   1:  PR[91,3] = PR[90,3] + 20.865;
   1:L PR[91] R[100]mm/sec CNT100;
   1:  PR[91,1] = PR[90,1] + -32.323;
   1:  PR[91,2] = PR[90,2] + 9.963;
   1:  PR[91,3] = PR[90,3] + 20.871;
   1:L PR[91] R[100]mm/sec CNT100;
   1:  PR[91,1] = PR[90,1] + -32.788;
   1:  PR[91,2] = PR[90,2] + 9.239;
   1:  PR[91,3] = PR[90,3] + 20.877;
   1:L PR[91] R[100]mm/sec CNT100;
   1:  PR[91,1] = PR[90,1] + -33.216;
   1:  PR[91,2] = PR[90,2] + 8.495;
   1:  PR[91,3] = PR[90,3] + 20.883;
   1:L PR[91] R[100]mm/sec CNT100;
   1:  PR[91,1] = PR[90,1] + -33.606;
   1:  PR[91,2] = PR[90,2] + 7.735;
   1:  PR[91,3] = PR[90,3] + 20.889;
   1:L PR[91] R[100]mm/sec CNT100;
   1:  PR[91,1] = PR[90,1] + -33.957;
   1:  PR[91,2] = PR[90,2] + 6.963;
   1:  PR[91,3] = PR[90,3] + 20.895;
   1:L PR[91] R[100]mm/sec CNT100;
   1:  PR[91,1] = PR[90,1] + -34.268;
   1:  PR[91,2] = PR[90,2] + 6.184;
   1:  PR[91,3] = PR[90,3] + 20.901;
   1:L PR[91] R[100]mm/sec CNT100;
   1:  PR[91,1] = PR[90,1] + -34.538;
   1:  PR[91,2] = PR[90,2] + 5.400;
   1:  PR[91,3] = PR[90,3] + 20.907;
   1:L PR[91] R[100]mm/sec CNT100;
   1:  PR[91,1] = PR[90,1] + -34.767;
   1:  PR[91,2] = PR[90,2] + 4.609;
   1:  PR[91,3] = PR[90,3] + 20.913;
   1:L PR[91] R[100]mm/sec CNT100;
   1:  PR[91,1] = PR[90,1] + -34.955;
   1:  PR[91,2] = PR[90,2] + 3.810;
   1:  PR[91,3] = PR[90,3] + 20.918;
   1:L PR[91] R[100]mm/sec CNT100;
   1:  PR[91,1] = PR[90,1] + -35.101;
   1:  PR[91,2] = PR[90,2] + 2.999;
   1:  PR[91,3] = PR[90,3] + 20.924;
   1:L PR[91] R[100]mm/sec CNT100;
   1:  PR[91,1] = PR[90,1] + -35.206;
   1:  PR[91,2] = PR[90,2] + 2.168;
   1:  PR[91,3] = PR[90,3] + 20.930;
   1:L PR[91] R[100]mm/sec CNT100;
   1:  PR[91,1] = PR[90,1] + -35.270;
   1:  PR[91,2] = PR[90,2] + 1.312;
   1:  PR[91,3] = PR[90,3] + 20.936;
   1:L PR[91] R[100]mm/sec CNT100;
   1:  PR[91,1] = PR[90,1] + -35.294;
   1:  PR[91,2] = PR[90,2] + 0.428;
   1:  PR[91,3] = PR[90,3] + 20.942;
   1:L PR[91] R[100]mm/sec CNT100;
   1:  PR[91,1] = PR[90,1] + -35.270;
   1:  PR[91,2] = PR[90,2] + -0.456;
   1:  PR[91,3] = PR[90,3] + 20.948;
   1:L PR[91] R[100]mm/sec CNT100;
   1:  PR[91,1] = PR[90,1] + -35.206;
   1:  PR[91,2] = PR[90,2] + -1.313;
   1:  PR[91,3] = PR[90,3] + 20.954;
   1:L PR[91] R[100]mm/sec CNT100;
   1:  PR[91,1] = PR[90,1] + -35.101;
   1:  PR[91,2] = PR[90,2] + -2.144;
   1:  PR[91,3] = PR[90,3] + 20.960;
   1:L PR[91] R[100]mm/sec CNT100;
   1:  PR[91,1] = PR[90,1] + -34.955;
   1:  PR[91,2] = PR[90,2] + -2.955;
   1:  PR[91,3] = PR[90,3] + 20.966;
   1:L PR[91] R[100]mm/sec CNT100;
   1:  PR[91,1] = PR[90,1] + -34.767;
   1:  PR[91,2] = PR[90,2] + -3.754;
   1:  PR[91,3] = PR[90,3] + 20.972;
   1:L PR[91] R[100]mm/sec CNT100;
   1:  PR[91,1] = PR[90,1] + -34.538;
   1:  PR[91,2] = PR[90,2] + -4.545;
   1:  PR[91,3] = PR[90,3] + 20.978;
   1:L PR[91] R[100]mm/sec CNT100;
   1:  PR[91,1] = PR[90,1] + -34.268;
   1:  PR[91,2] = PR[90,2] + -5.329;
   1:  PR[91,3] = PR[90,3] + 20.984;
   1:L PR[91] R[100]mm/sec CNT100;
   1:  PR[91,1] = PR[90,1] + -33.956;
   1:  PR[91,2] = PR[90,2] + -6.108;
   1:  PR[91,3] = PR[90,3] + 20.989;
   1:L PR[91] R[100]mm/sec CNT100;
   1:  PR[91,1] = PR[90,1] + -33.606;
   1:  PR[91,2] = PR[90,2] + -6.880;
   1:  PR[91,3] = PR[90,3] + 20.995;
   1:L PR[91] R[100]mm/sec CNT100;
   1:  PR[91,1] = PR[90,1] + -33.216;
   1:  PR[91,2] = PR[90,2] + -7.640;
   1:  PR[91,3] = PR[90,3] + 21.001;
   1:L PR[91] R[100]mm/sec CNT100;
   1:  PR[91,1] = PR[90,1] + -32.788;
   1:  PR[91,2] = PR[90,2] + -8.384;
   1:  PR[91,3] = PR[90,3] + 21.007;
   1:L PR[91] R[100]mm/sec CNT100;
   1:  PR[91,1] = PR[90,1] + -32.323;
   1:  PR[91,2] = PR[90,2] + -9.108;
   1:  PR[91,3] = PR[90,3] + 21.013;
   1:L PR[91] R[100]mm/sec CNT100;
   1:  PR[91,1] = PR[90,1] + -31.822;
   1:  PR[91,2] = PR[90,2] + -9.809;
   1:  PR[91,3] = PR[90,3] + 21.019;
   1:L PR[91] R[100]mm/sec CNT100;
   1:  PR[91,1] = PR[90,1] + -31.285;
   1:  PR[91,2] = PR[90,2] + -10.485;
   1:  PR[91,3] = PR[90,3] + 21.026;
   1:L PR[91] R[100]mm/sec CNT100;
   1:  PR[91,1] = PR[90,1] + -30.715;
   1:  PR[91,2] = PR[90,2] + -11.134;
   1:  PR[91,3] = PR[90,3] + 21.032;
   1:L PR[91] R[100]mm/sec CNT100;
   1:  PR[91,1] = PR[90,1] + -30.107;
   1:  PR[91,2] = PR[90,2] + -11.756;
   1:  PR[91,3] = PR[90,3] + 21.038;
   1:L PR[91] R[100]mm/sec CNT100;
   1:  PR[91,1] = PR[90,1] + -29.466;
   1:  PR[91,2] = PR[90,2] + -12.350;
   1:  PR[91,3] = PR[90,3] + 21.044;
   1:L PR[91] R[100]mm/sec CNT100;
   1:  PR[91,1] = PR[90,1] + -28.795;
   1:  PR[91,2] = PR[90,2] + -12.914;
   1:  PR[91,3] = PR[90,3] + 21.050;
   1:L PR[91] R[100]mm/sec CNT100;
   1:  PR[91,1] = PR[90,1] + -28.093;
   1:  PR[91,2] = PR[90,2] + -13.447;
   1:  PR[91,3] = PR[90,3] + 21.056;
   1:L PR[91] R[100]mm/sec CNT100;
   1:  PR[91,1] = PR[90,1] + -27.361;
   1:  PR[91,2] = PR[90,2] + -13.949;
   1:  PR[91,3] = PR[90,3] + 21.062;
   1:L PR[91] R[100]mm/sec CNT100;
   1:  PR[91,1] = PR[90,1] + -27.042;
   1:  PR[91,2] = PR[90,2] + -14.147;
   1:  PR[91,3] = PR[90,3] + 21.069;
   1:L PR[91] R[100]mm/sec CNT100;
   1:  PR[91,1] = PR[90,1] + -26.605;
   1:  PR[91,2] = PR[90,2] + -14.416;
   1:  PR[91,3] = PR[90,3] + 21.071;
   1:L PR[91] R[100]mm/sec CNT100;
   1:  PR[91,1] = PR[90,1] + -25.820;
   1:  PR[91,2] = PR[90,2] + -14.850;
   1:  PR[91,3] = PR[90,3] + 21.075;
   1:L PR[91] R[100]mm/sec CNT100;
   1:  PR[91,1] = PR[90,1] + -25.013;
   1:  PR[91,2] = PR[90,2] + -15.247;
   1:  PR[91,3] = PR[90,3] + 21.081;
   1:L PR[91] R[100]mm/sec CNT100;
   1:  PR[91,1] = PR[90,1] + -24.202;
   1:  PR[91,2] = PR[90,2] + -15.599;
   1:  PR[91,3] = PR[90,3] + 21.087;
   1:L PR[91] R[100]mm/sec CNT100;
   1:  PR[91,1] = PR[90,1] + -23.226;
   1:  PR[91,2] = PR[90,2] + -15.963;
   1:  PR[91,3] = PR[90,3] + 21.094;
   1:L PR[91] R[100]mm/sec CNT100;
   1:  PR[91,1] = PR[90,1] + -22.273;
   1:  PR[91,2] = PR[90,2] + -16.262;
   1:  PR[91,3] = PR[90,3] + 21.101;
   1:L PR[91] R[100]mm/sec CNT100;
   1:  PR[91,1] = PR[90,1] + -21.780;
   1:  PR[91,2] = PR[90,2] + -16.396;
   1:  PR[91,3] = PR[90,3] + 21.108;
   1:L PR[91] R[100]mm/sec CNT100;
   1:  PR[91,1] = PR[90,1] + -20.956;
   1:  PR[91,2] = PR[90,2] + -16.588;
   1:  PR[91,3] = PR[90,3] + 21.112;
   1:L PR[91] R[100]mm/sec CNT100;
   1:  PR[91,1] = PR[90,1] + -20.130;
   1:  PR[91,2] = PR[90,2] + -16.744;
   1:  PR[91,3] = PR[90,3] + 21.118;
   1:L PR[91] R[100]mm/sec CNT100;
   1:  PR[91,1] = PR[90,1] + -19.301;
   1:  PR[91,2] = PR[90,2] + -16.862;
   1:  PR[91,3] = PR[90,3] + 21.124;
   1:L PR[91] R[100]mm/sec CNT100;
   1:  PR[91,1] = PR[90,1] + -18.404;
   1:  PR[91,2] = PR[90,2] + -16.950;
   1:  PR[91,3] = PR[90,3] + 21.129;
   1:L PR[91] R[100]mm/sec CNT100;
   1:  PR[91,1] = PR[90,1] + -17.474;
   1:  PR[91,2] = PR[90,2] + -16.997;
   1:  PR[91,3] = PR[90,3] + 21.136;
   1:L PR[91] R[100]mm/sec CNT100;
   1:  PR[91,1] = PR[90,1] + -16.945;
   1:  PR[91,2] = PR[90,2] + -17.001;
   1:  PR[91,3] = PR[90,3] + 21.142;
   1:L PR[91] R[100]mm/sec CNT100;
   1:  PR[91,1] = PR[90,1] + -16.543;
   1:  PR[91,3] = PR[90,3] + 21.146;
   1:L PR[91] R[100]mm/sec CNT100;
   1:  PR[91,1] = PR[90,1] + -15.605;
   1:  PR[91,2] = PR[90,2] + -16.959;
   1:  PR[91,3] = PR[90,3] + 21.149;
   1:L PR[91] R[100]mm/sec CNT100;
   1:  PR[91,1] = PR[90,1] + -14.668;
   1:  PR[91,2] = PR[90,2] + -16.872;
   1:  PR[91,3] = PR[90,3] + 21.156;
   1:L PR[91] R[100]mm/sec CNT100;
   1:  PR[91,1] = PR[90,1] + -13.745;
   1:  PR[91,2] = PR[90,2] + -16.743;
   1:  PR[91,3] = PR[90,3] + 21.162;
   1:L PR[91] R[100]mm/sec CNT100;
   1:  PR[91,1] = PR[90,1] + -12.925;
   1:  PR[91,2] = PR[90,2] + -16.592;
   1:  PR[91,3] = PR[90,3] + 21.169;
   1:L PR[91] R[100]mm/sec CNT100;
   1:  PR[91,1] = PR[90,1] + -11.875;
   1:  PR[91,2] = PR[90,2] + -16.344;
   1:  PR[91,3] = PR[90,3] + 21.175;
   1:L PR[91] R[100]mm/sec CNT100;
   1:  PR[91,1] = PR[90,1] + -11.166;
   1:  PR[91,2] = PR[90,2] + -16.141;
   1:  PR[91,3] = PR[90,3] + 21.182;
   1:L PR[91] R[100]mm/sec CNT100;
   1:  PR[91,1] = PR[90,1] + -10.545;
   1:  PR[91,2] = PR[90,2] + -15.938;
   1:  PR[91,3] = PR[90,3] + 21.187;
   1:L PR[91] R[100]mm/sec CNT100;
   1:  PR[91,1] = PR[90,1] + -9.970;
   1:  PR[91,2] = PR[90,2] + -15.731;
   1:  PR[91,3] = PR[90,3] + 21.192;
   1:L PR[91] R[100]mm/sec CNT100;
   1:  PR[91,1] = PR[90,1] + -9.341;
   1:  PR[91,2] = PR[90,2] + -15.480;
   1:  PR[91,3] = PR[90,3] + 21.196;
   1:L PR[91] R[100]mm/sec CNT100;
   1:  PR[91,1] = PR[90,1] + -8.803;
   1:  PR[91,2] = PR[90,2] + -15.246;
   1:  PR[91,3] = PR[90,3] + 21.201;
   1:L PR[91] R[100]mm/sec CNT100;
   1:  PR[91,1] = PR[90,1] + -8.183;
   1:  PR[91,2] = PR[90,2] + -14.951;
   1:  PR[91,3] = PR[90,3] + 21.205;
   1:L PR[91] R[100]mm/sec CNT100;
   1:  PR[91,1] = PR[90,1] + -7.109;
   1:  PR[91,2] = PR[90,2] + -14.372;
   1:  PR[91,3] = PR[90,3] + 21.210;
   1:L PR[91] R[100]mm/sec CNT100;
   1:  PR[91,1] = PR[90,1] + -6.488;
   1:  PR[91,2] = PR[90,2] + -13.995;
   1:  PR[91,3] = PR[90,3] + 21.219;
   1:L PR[91] R[100]mm/sec CNT100;
   1:  PR[91,1] = PR[90,1] + -5.527;
   1:  PR[91,2] = PR[90,2] + -13.342;
   1:  PR[91,3] = PR[90,3] + 21.224;
   1:L PR[91] R[100]mm/sec CNT100;
   1:  PR[91,1] = PR[90,1] + -4.920;
   1:  PR[91,2] = PR[90,2] + -12.883;
   1:  PR[91,3] = PR[90,3] + 21.232;
   1:L PR[91] R[100]mm/sec CNT100;
   1:  PR[91,1] = PR[90,1] + -4.075;
   1:  PR[91,2] = PR[90,2] + -12.171;
   1:  PR[91,3] = PR[90,3] + 21.237;
   1:L PR[91] R[100]mm/sec CNT100;
   1:  PR[91,1] = PR[90,1] + -3.306;
   1:  PR[91,2] = PR[90,2] + -11.437;
   1:  PR[91,3] = PR[90,3] + 21.245;
   1:L PR[91] R[100]mm/sec CNT100;
   1:  PR[91,1] = PR[90,1] + -2.752;
   1:  PR[91,2] = PR[90,2] + -10.852;
   1:  PR[91,3] = PR[90,3] + 21.253;
   1:L PR[91] R[100]mm/sec CNT100;
   1:  PR[91,1] = PR[90,1] + -2.351;
   1:  PR[91,2] = PR[90,2] + -10.384;
   1:  PR[91,3] = PR[90,3] + 21.258;
   1:L PR[91] R[100]mm/sec CNT100;
   1:  PR[91,1] = PR[90,1] + -2.018;
   1:  PR[91,2] = PR[90,2] + -10.037;
   1:  PR[91,3] = PR[90,3] + 21.263;
   1:L PR[91] R[100]mm/sec CNT100;
   1:  PR[91,1] = PR[90,1] + -1.614;
   1:  PR[91,2] = PR[90,2] + -9.738;
   1:  PR[91,3] = PR[90,3] + 21.266;
   1:L PR[91] R[100]mm/sec CNT100;
   1:  PR[91,1] = PR[90,1] + -1.170;
   1:  PR[91,2] = PR[90,2] + -9.512;
   1:  PR[91,3] = PR[90,3] + 21.269;
   1:L PR[91] R[100]mm/sec CNT100;
   1:  PR[91,1] = PR[90,1] + -0.694;
   1:  PR[91,2] = PR[90,2] + -9.365;
   1:  PR[91,3] = PR[90,3] + 21.273;
   1:L PR[91] R[100]mm/sec CNT100;
   1:  PR[91,1] = PR[90,1] + -0.199;
   1:  PR[91,2] = PR[90,2] + -9.306;
   1:  PR[91,3] = PR[90,3] + 21.276;
   1:L PR[91] R[100]mm/sec CNT100;
   1:  PR[91] = PR[90];
   1:  PR[91,1] = PR[90,1] + 0.421;
   1:  PR[91,2] = PR[90,2] + -10.128;
   1:  PR[91,3] = PR[90,3] + 22.610;
   1:L PR[91] R[100]mm/sec CNT100;
   1:  PR[91,1] = PR[90,1] + 0.906;
   1:  PR[91,2] = PR[90,2] + -10.267;
   1:  PR[91,3] = PR[90,3] + 21.284;
   1:L PR[91] R[100]mm/sec CNT100;
   1:  PR[91,1] = PR[90,1] + 1.365;
   1:  PR[91,2] = PR[90,2] + -10.492;
   1:  PR[91,3] = PR[90,3] + 21.287;
   1:L PR[91] R[100]mm/sec CNT100;
   1:  PR[91,1] = PR[90,1] + 1.785;
   1:  PR[91,2] = PR[90,2] + -10.796;
   1:  PR[91,3] = PR[90,3] + 21.291;
   1:L PR[91] R[100]mm/sec CNT100;
   1:  PR[91,1] = PR[90,1] + 2.627;
   1:  PR[91,2] = PR[90,2] + -11.664;
   1:  PR[91,3] = PR[90,3] + 21.294;
   1:L PR[91] R[100]mm/sec CNT100;
   1:  PR[91,1] = PR[90,1] + 3.330;
   1:  PR[91,2] = PR[90,2] + -12.323;
   1:  PR[91,3] = PR[90,3] + 21.303;
   1:L PR[91] R[100]mm/sec CNT100;
   1:  PR[91,1] = PR[90,1] + 4.018;
   1:  PR[91,2] = PR[90,2] + -12.904;
   1:  PR[91,3] = PR[90,3] + 21.310;
   1:L PR[91] R[100]mm/sec CNT100;
   1:  PR[91,1] = PR[90,1] + 4.792;
   1:  PR[91,2] = PR[90,2] + -13.492;
   1:  PR[91,3] = PR[90,3] + 21.316;
   1:L PR[91] R[100]mm/sec CNT100;
   1:  PR[91,1] = PR[90,1] + 5.634;
   1:  PR[91,2] = PR[90,2] + -14.062;
   1:  PR[91,3] = PR[90,3] + 21.323;
   1:L PR[91] R[100]mm/sec CNT100;
   1:  PR[91,1] = PR[90,1] + 6.385;
   1:  PR[91,2] = PR[90,2] + -14.517;
   1:  PR[91,3] = PR[90,3] + 21.331;
   1:L PR[91] R[100]mm/sec CNT100;
   1:  PR[91,1] = PR[90,1] + 7.324;
   1:  PR[91,2] = PR[90,2] + -15.021;
   1:  PR[91,3] = PR[90,3] + 21.337;
   1:L PR[91] R[100]mm/sec CNT100;
   1:  PR[91,1] = PR[90,1] + 8.080;
   1:  PR[91,2] = PR[90,2] + -15.379;
   1:  PR[91,3] = PR[90,3] + 21.344;
   1:L PR[91] R[100]mm/sec CNT100;
   1:  PR[91,1] = PR[90,1] + 9.117;
   1:  PR[91,2] = PR[90,2] + -15.808;
   1:  PR[91,3] = PR[90,3] + 21.350;
   1:L PR[91] R[100]mm/sec CNT100;
   1:  PR[91,1] = PR[90,1] + 9.860;
   1:  PR[91,2] = PR[90,2] + -16.074;
   1:  PR[91,3] = PR[90,3] + 21.358;
   1:L PR[91] R[100]mm/sec CNT100;
   1:  PR[91,1] = PR[90,1] + 10.982;
   1:  PR[91,2] = PR[90,2] + -16.413;
   1:  PR[91,3] = PR[90,3] + 21.364;
   1:L PR[91] R[100]mm/sec CNT100;
   1:  PR[91,1] = PR[90,1] + 12.190;
   1:  PR[91,2] = PR[90,2] + -16.698;
   1:  PR[91,3] = PR[90,3] + 21.372;
   1:L PR[91] R[100]mm/sec CNT100;
   1:  PR[91,1] = PR[90,1] + 12.901;
   1:  PR[91,2] = PR[90,2] + -16.830;
   1:  PR[91,3] = PR[90,3] + 21.381;
   1:L PR[91] R[100]mm/sec CNT100;
   1:  PR[91,1] = PR[90,1] + 13.574;
   1:  PR[91,2] = PR[90,2] + -16.929;
   1:  PR[91,3] = PR[90,3] + 21.386;
   1:L PR[91] R[100]mm/sec CNT100;
   1:  PR[91,1] = PR[90,1] + 14.840;
   1:  PR[91,2] = PR[90,2] + -17.053;
   1:  PR[91,3] = PR[90,3] + 21.391;
   1:L PR[91] R[100]mm/sec CNT100;
   1:  PR[91,1] = PR[90,1] + 16.006;
   1:  PR[91,2] = PR[90,2] + -17.097;
   1:  PR[91,3] = PR[90,3] + 21.400;
   1:L PR[91] R[100]mm/sec CNT100;
   1:  PR[91,1] = PR[90,1] + 16.711;
   1:  PR[91,2] = PR[90,2] + -17.091;
   1:  PR[91,3] = PR[90,3] + 21.409;
   1:L PR[91] R[100]mm/sec CNT100;
   1:  PR[91,1] = PR[90,1] + 17.506;
   1:  PR[91,2] = PR[90,2] + -17.054;
   1:  PR[91,3] = PR[90,3] + 21.414;
   1:L PR[91] R[100]mm/sec CNT100;
   1:  PR[91,1] = PR[90,1] + 18.499;
   1:  PR[91,2] = PR[90,2] + -16.963;
   1:  PR[91,3] = PR[90,3] + 21.419;
   1:L PR[91] R[100]mm/sec CNT100;
   1:  PR[91,1] = PR[90,1] + 19.377;
   1:  PR[91,2] = PR[90,2] + -16.840;
   1:  PR[91,3] = PR[90,3] + 21.426;
   1:L PR[91] R[100]mm/sec CNT100;
   1:  PR[91,1] = PR[90,1] + 20.291;
   1:  PR[91,2] = PR[90,2] + -16.668;
   1:  PR[91,3] = PR[90,3] + 21.433;
   1:L PR[91] R[100]mm/sec CNT100;
   1:  PR[91,1] = PR[90,1] + 21.192;
   1:  PR[91,2] = PR[90,2] + -16.455;
   1:  PR[91,3] = PR[90,3] + 21.439;
   1:L PR[91] R[100]mm/sec CNT100;
   1:  PR[91,1] = PR[90,1] + 22.077;
   1:  PR[91,2] = PR[90,2] + -16.200;
   1:  PR[91,3] = PR[90,3] + 21.446;
   1:L PR[91] R[100]mm/sec CNT100;
   1:  PR[91,1] = PR[90,1] + 22.945;
   1:  PR[91,2] = PR[90,2] + -15.905;
   1:  PR[91,3] = PR[90,3] + 21.453;
   1:L PR[91] R[100]mm/sec CNT100;
   1:  PR[91,1] = PR[90,1] + 23.794;
   1:  PR[91,2] = PR[90,2] + -15.572;
   1:  PR[91,3] = PR[90,3] + 21.459;
   1:L PR[91] R[100]mm/sec CNT100;
   1:  PR[91,1] = PR[90,1] + 24.595;
   1:  PR[91,2] = PR[90,2] + -15.214;
   1:  PR[91,3] = PR[90,3] + 21.466;
   1:L PR[91] R[100]mm/sec CNT100;
   1:  PR[91,1] = PR[90,1] + 25.352;
   1:  PR[91,2] = PR[90,2] + -14.833;
   1:  PR[91,3] = PR[90,3] + 21.472;
   1:L PR[91] R[100]mm/sec CNT100;
   1:  PR[91,1] = PR[90,1] + 26.092;
   1:  PR[91,2] = PR[90,2] + -14.417;
   1:  PR[91,3] = PR[90,3] + 21.478;
   1:L PR[91] R[100]mm/sec CNT100;
   1:  PR[91,1] = PR[90,1] + 26.814;
   1:  PR[91,2] = PR[90,2] + -13.968;
   1:  PR[91,3] = PR[90,3] + 21.484;
   1:L PR[91] R[100]mm/sec CNT100;
   1:  PR[91,1] = PR[90,1] + 27.516;
   1:  PR[91,2] = PR[90,2] + -13.485;
   1:  PR[91,3] = PR[90,3] + 21.490;
   1:L PR[91] R[100]mm/sec CNT100;
   1:  PR[91,1] = PR[90,1] + 28.196;
   1:  PR[91,2] = PR[90,2] + -12.969;
   1:  PR[91,3] = PR[90,3] + 21.496;
   1:L PR[91] R[100]mm/sec CNT100;
   1:  PR[91,1] = PR[90,1] + 28.852;
   1:  PR[91,2] = PR[90,2] + -12.420;
   1:  PR[91,3] = PR[90,3] + 21.502;
   1:L PR[91] R[100]mm/sec CNT100;
   1:  PR[91,1] = PR[90,1] + 29.481;
   1:  PR[91,2] = PR[90,2] + -11.840;
   1:  PR[91,3] = PR[90,3] + 21.508;
   1:L PR[91] R[100]mm/sec CNT100;
   1:  PR[91,1] = PR[90,1] + 30.083;
   1:  PR[91,2] = PR[90,2] + -11.228;
   1:  PR[91,3] = PR[90,3] + 21.514;
   1:L PR[91] R[100]mm/sec CNT100;
   1:  PR[91,1] = PR[90,1] + 30.665;
   1:  PR[91,2] = PR[90,2] + -10.571;
   1:  PR[91,3] = PR[90,3] + 21.521;
   1:L PR[91] R[100]mm/sec CNT100;
   1:  PR[91,1] = PR[90,1] + 31.212;
   1:  PR[91,2] = PR[90,2] + -9.887;
   1:  PR[91,3] = PR[90,3] + 21.527;
   1:L PR[91] R[100]mm/sec CNT100;
   1:  PR[91,1] = PR[90,1] + 31.723;
   1:  PR[91,2] = PR[90,2] + -9.178;
   1:  PR[91,3] = PR[90,3] + 21.533;
   1:L PR[91] R[100]mm/sec CNT100;
   1:  PR[91,1] = PR[90,1] + 32.197;
   1:  PR[91,2] = PR[90,2] + -8.448;
   1:  PR[91,3] = PR[90,3] + 21.539;
   1:L PR[91] R[100]mm/sec CNT100;
   1:  PR[91,1] = PR[90,1] + 32.633;
   1:  PR[91,2] = PR[90,2] + -7.699;
   1:  PR[91,3] = PR[90,3] + 21.545;
   1:L PR[91] R[100]mm/sec CNT100;
   1:  PR[91,1] = PR[90,1] + 33.030;
   1:  PR[91,2] = PR[90,2] + -6.937;
   1:  PR[91,3] = PR[90,3] + 21.552;
   1:L PR[91] R[100]mm/sec CNT100;
   1:  PR[91,1] = PR[90,1] + 33.388;
   1:  PR[91,2] = PR[90,2] + -6.164;
   1:  PR[91,3] = PR[90,3] + 21.558;
   1:L PR[91] R[100]mm/sec CNT100;
   1:  PR[91,1] = PR[90,1] + 33.704;
   1:  PR[91,2] = PR[90,2] + -5.385;
   1:  PR[91,3] = PR[90,3] + 21.564;
   1:L PR[91] R[100]mm/sec CNT100;
   1:  PR[91,1] = PR[90,1] + 33.979;
   1:  PR[91,2] = PR[90,2] + -4.600;
   1:  PR[91,3] = PR[90,3] + 21.570;
   1:L PR[91] R[100]mm/sec CNT100;
   1:  PR[91,1] = PR[90,1] + 34.212;
   1:  PR[91,2] = PR[90,2] + -3.806;
   1:  PR[91,3] = PR[90,3] + 21.576;
   1:L PR[91] R[100]mm/sec CNT100;
   1:  PR[91,1] = PR[90,1] + 34.403;
   1:  PR[91,2] = PR[90,2] + -3.001;
   1:  PR[91,3] = PR[90,3] + 21.582;
   1:L PR[91] R[100]mm/sec CNT100;
   1:  PR[91,1] = PR[90,1] + 34.552;
   1:  PR[91,2] = PR[90,2] + -2.180;
   1:  PR[91,3] = PR[90,3] + 21.588;
   1:L PR[91] R[100]mm/sec CNT100;
   1:  PR[91,1] = PR[90,1] + 34.659;
   1:  PR[91,2] = PR[90,2] + -1.338;
   1:  PR[91,3] = PR[90,3] + 21.594;
   1:L PR[91] R[100]mm/sec CNT100;
   1:  PR[91,1] = PR[90,1] + 34.724;
   1:  PR[91,2] = PR[90,2] + -0.470;
   1:  PR[91,3] = PR[90,3] + 21.600;
   1:L PR[91] R[100]mm/sec CNT100;
   1:  PR[91,1] = PR[90,1] + 34.745;
   1:  PR[91,2] = PR[90,2] + 0.428;
   1:  PR[91,3] = PR[90,3] + 21.606;
   1:L PR[91] R[100]mm/sec CNT100;
   1:  PR[91,1] = PR[90,1] + 34.724;
   1:  PR[91,2] = PR[90,2] + 1.325;
   1:  PR[91,3] = PR[90,3] + 21.612;
   1:L PR[91] R[100]mm/sec CNT100;
   1:  PR[91,1] = PR[90,1] + 34.659;
   1:  PR[91,2] = PR[90,2] + 2.193;
   1:  PR[91,3] = PR[90,3] + 21.619;
   1:L PR[91] R[100]mm/sec CNT100;
   1:  PR[91,1] = PR[90,1] + 34.552;
   1:  PR[91,2] = PR[90,2] + 3.035;
   1:  PR[91,3] = PR[90,3] + 21.625;
   1:L PR[91] R[100]mm/sec CNT100;
   1:  PR[91,1] = PR[90,1] + 34.403;
   1:  PR[91,2] = PR[90,2] + 3.856;
   1:  PR[91,3] = PR[90,3] + 21.631;
   1:L PR[91] R[100]mm/sec CNT100;
   1:  PR[91,1] = PR[90,1] + 34.212;
   1:  PR[91,2] = PR[90,2] + 4.661;
   1:  PR[91,3] = PR[90,3] + 21.637;
   1:L PR[91] R[100]mm/sec CNT100;
   1:  PR[91,1] = PR[90,1] + 33.979;
   1:  PR[91,2] = PR[90,2] + 5.455;
   1:  PR[91,3] = PR[90,3] + 21.643;
   1:L PR[91] R[100]mm/sec CNT100;
   1:  PR[91,1] = PR[90,1] + 33.704;
   1:  PR[91,2] = PR[90,2] + 6.241;
   1:  PR[91,3] = PR[90,3] + 21.649;
   1:L PR[91] R[100]mm/sec CNT100;
   1:  PR[91,1] = PR[90,1] + 33.388;
   1:  PR[91,2] = PR[90,2] + 7.019;
   1:  PR[91,3] = PR[90,3] + 21.655;
   1:L PR[91] R[100]mm/sec CNT100;
   1:  PR[91,1] = PR[90,1] + 33.030;
   1:  PR[91,2] = PR[90,2] + 7.792;
   1:  PR[91,3] = PR[90,3] + 21.661;
   1:L PR[91] R[100]mm/sec CNT100;
   1:  PR[91,1] = PR[90,1] + 32.633;
   1:  PR[91,2] = PR[90,2] + 8.554;
   1:  PR[91,3] = PR[90,3] + 21.667;
   1:L PR[91] R[100]mm/sec CNT100;
   1:  PR[91,1] = PR[90,1] + 32.197;
   1:  PR[91,2] = PR[90,2] + 9.303;
   1:  PR[91,3] = PR[90,3] + 21.673;
   1:L PR[91] R[100]mm/sec CNT100;
   1:  PR[91,1] = PR[90,1] + 31.723;
   1:  PR[91,2] = PR[90,2] + 10.033;
   1:  PR[91,3] = PR[90,3] + 21.679;
   1:L PR[91] R[100]mm/sec CNT100;
   1:  PR[91,1] = PR[90,1] + 31.212;
   1:  PR[91,2] = PR[90,2] + 10.742;
   1:  PR[91,3] = PR[90,3] + 21.685;
   1:L PR[91] R[100]mm/sec CNT100;
   1:  PR[91,1] = PR[90,1] + 30.665;
   1:  PR[91,2] = PR[90,2] + 11.426;
   1:  PR[91,3] = PR[90,3] + 21.691;
   1:L PR[91] R[100]mm/sec CNT100;
   1:  PR[91,1] = PR[90,1] + 30.081;
   1:  PR[91,2] = PR[90,2] + 12.086;
   1:  PR[91,3] = PR[90,3] + 21.698;
   1:L PR[91] R[100]mm/sec CNT100;
   1:  PR[91,1] = PR[90,1] + 29.481;
   1:  PR[91,2] = PR[90,2] + 12.695;
   1:  PR[91,3] = PR[90,3] + 21.704;
   1:L PR[91] R[100]mm/sec CNT100;
   1:  PR[91,1] = PR[90,1] + 28.852;
   1:  PR[91,2] = PR[90,2] + 13.276;
   1:  PR[91,3] = PR[90,3] + 21.710;
   1:L PR[91] R[100]mm/sec CNT100;
   1:  PR[91,1] = PR[90,1] + 28.196;
   1:  PR[91,2] = PR[90,2] + 13.824;
   1:  PR[91,3] = PR[90,3] + 21.716;
   1:L PR[91] R[100]mm/sec CNT100;
   1:  PR[91,1] = PR[90,1] + 27.515;
   1:  PR[91,2] = PR[90,2] + 14.341;
   1:  PR[91,3] = PR[90,3] + 21.722;
   1:L PR[91] R[100]mm/sec CNT100;
   1:  PR[91,1] = PR[90,1] + 27.184;
   1:  PR[91,2] = PR[90,2] + 14.571;
   1:  PR[91,3] = PR[90,3] + 21.728;
   1:L PR[91] R[100]mm/sec CNT100;
   1:  PR[91,1] = PR[90,1] + 26.815;
   1:  PR[91,2] = PR[90,2] + 14.822;
   1:  PR[91,3] = PR[90,3] + 21.731;
   1:L PR[91] R[100]mm/sec CNT100;
   1:  PR[91,1] = PR[90,1] + 26.092;
   1:  PR[91,2] = PR[90,2] + 15.272;
   1:  PR[91,3] = PR[90,3] + 21.734;
   1:L PR[91] R[100]mm/sec CNT100;
   1:  PR[91,1] = PR[90,1] + 25.352;
   1:  PR[91,2] = PR[90,2] + 15.688;
   1:  PR[91,3] = PR[90,3] + 21.740;
   1:L PR[91] R[100]mm/sec CNT100;
   1:  PR[91,1] = PR[90,1] + 24.595;
   1:  PR[91,2] = PR[90,2] + 16.069;
   1:  PR[91,3] = PR[90,3] + 21.746;
   1:L PR[91] R[100]mm/sec CNT100;
   1:  PR[91,1] = PR[90,1] + 23.794;
   1:  PR[91,2] = PR[90,2] + 16.428;
   1:  PR[91,3] = PR[90,3] + 21.752;
   1:L PR[91] R[100]mm/sec CNT100;
   1:  PR[91,1] = PR[90,1] + 22.944;
   1:  PR[91,2] = PR[90,2] + 16.761;
   1:  PR[91,3] = PR[90,3] + 21.759;
   1:L PR[91] R[100]mm/sec CNT100;
   1:  PR[91,1] = PR[90,1] + 22.377;
   1:  PR[91,2] = PR[90,2] + 16.955;
   1:  PR[91,3] = PR[90,3] + 21.765;
   1:L PR[91] R[100]mm/sec CNT100;
   1:  PR[91,1] = PR[90,1] + 22.078;
   1:  PR[91,2] = PR[90,2] + 17.055;
   1:  PR[91,3] = PR[90,3] + 21.770;
   1:L PR[91] R[100]mm/sec CNT100;
   1:  PR[91,1] = PR[90,1] + 21.194;
   1:  PR[91,2] = PR[90,2] + 17.309;
   1:  PR[91,3] = PR[90,3] + 21.772;
   1:L PR[91] R[100]mm/sec CNT100;
   1:  PR[91,1] = PR[90,1] + 20.105;
   1:  PR[91,2] = PR[90,2] + 17.560;
   1:  PR[91,3] = PR[90,3] + 21.778;
   1:L PR[91] R[100]mm/sec CNT100;
   1:  PR[91,1] = PR[90,1] + 19.377;
   1:  PR[91,2] = PR[90,2] + 17.695;
   1:  PR[91,3] = PR[90,3] + 21.786;
   1:L PR[91] R[100]mm/sec CNT100;
   1:  PR[91,1] = PR[90,1] + 18.499;
   1:  PR[91,2] = PR[90,2] + 17.818;
   1:  PR[91,3] = PR[90,3] + 21.792;
   1:L PR[91] R[100]mm/sec CNT100;
   1:  PR[91,1] = PR[90,1] + 17.506;
   1:  PR[91,2] = PR[90,2] + 17.909;
   1:  PR[91,3] = PR[90,3] + 21.798;
   1:L PR[91] R[100]mm/sec CNT100;
   1:  PR[91,1] = PR[90,1] + 16.710;
   1:  PR[91,2] = PR[90,2] + 17.946;
   1:  PR[91,3] = PR[90,3] + 21.805;
   1:L PR[91] R[100]mm/sec CNT100;
   1:  PR[91,1] = PR[90,1] + 16.006;
   1:  PR[91,2] = PR[90,2] + 17.952;
   1:  PR[91,3] = PR[90,3] + 21.811;
   1:L PR[91] R[100]mm/sec CNT100;
   1:  PR[91,1] = PR[90,1] + 14.836;
   1:  PR[91,2] = PR[90,2] + 17.908;
   1:  PR[91,3] = PR[90,3] + 21.816;
   1:L PR[91] R[100]mm/sec CNT100;
   1:  PR[91,1] = PR[90,1] + 14.180;
   1:  PR[91,2] = PR[90,2] + 17.854;
   1:  PR[91,3] = PR[90,3] + 21.824;
   1:L PR[91] R[100]mm/sec CNT100;
   1:  PR[91,1] = PR[90,1] + 13.579;
   1:  PR[91,2] = PR[90,2] + 17.785;
   1:  PR[91,3] = PR[90,3] + 21.829;
   1:L PR[91] R[100]mm/sec CNT100;
   1:  PR[91,1] = PR[90,1] + 12.901;
   1:  PR[91,2] = PR[90,2] + 17.685;
   1:  PR[91,3] = PR[90,3] + 21.833;
   1:L PR[91] R[100]mm/sec CNT100;
   1:  PR[91,1] = PR[90,1] + 12.184;
   1:  PR[91,2] = PR[90,2] + 17.552;
   1:  PR[91,3] = PR[90,3] + 21.838;
   1:L PR[91] R[100]mm/sec CNT100;
   1:  PR[91,1] = PR[90,1] + 11.707;
   1:  PR[91,2] = PR[90,2] + 17.449;
   1:  PR[91,3] = PR[90,3] + 21.843;
   1:L PR[91] R[100]mm/sec CNT100;
   1:  PR[91,1] = PR[90,1] + 10.579;
   1:  PR[91,2] = PR[90,2] + 17.153;
   1:  PR[91,3] = PR[90,3] + 21.847;
   1:L PR[91] R[100]mm/sec CNT100;
   1:  PR[91,1] = PR[90,1] + 9.862;
   1:  PR[91,2] = PR[90,2] + 16.930;
   1:  PR[91,3] = PR[90,3] + 21.855;
   1:L PR[91] R[100]mm/sec CNT100;
   1:  PR[91,1] = PR[90,1] + 9.115;
   1:  PR[91,2] = PR[90,2] + 16.663;
   1:  PR[91,3] = PR[90,3] + 21.860;
   1:L PR[91] R[100]mm/sec CNT100;
   1:  PR[91,1] = PR[90,1] + 8.342;
   1:  PR[91,2] = PR[90,2] + 16.348;
   1:  PR[91,3] = PR[90,3] + 21.866;
   1:L PR[91] R[100]mm/sec CNT100;
   1:  PR[91,1] = PR[90,1] + 7.322;
   1:  PR[91,2] = PR[90,2] + 15.875;
   1:  PR[91,3] = PR[90,3] + 21.872;
   1:L PR[91] R[100]mm/sec CNT100;
   1:  PR[91,1] = PR[90,1] + 6.384;
   1:  PR[91,2] = PR[90,2] + 15.372;
   1:  PR[91,3] = PR[90,3] + 21.880;
   1:L PR[91] R[100]mm/sec CNT100;
   1:  PR[91,1] = PR[90,1] + 5.632;
   1:  PR[91,2] = PR[90,2] + 14.917;
   1:  PR[91,3] = PR[90,3] + 21.888;
   1:L PR[91] R[100]mm/sec CNT100;
   1:  PR[91,1] = PR[90,1] + 4.871;
   1:  PR[91,2] = PR[90,2] + 14.403;
   1:  PR[91,3] = PR[90,3] + 21.894;
   1:L PR[91] R[100]mm/sec CNT100;
   1:  PR[91,1] = PR[90,1] + 4.059;
   1:  PR[91,2] = PR[90,2] + 13.793;
   1:  PR[91,3] = PR[90,3] + 21.900;
   1:L PR[91] R[100]mm/sec CNT100;
   1:  PR[91,1] = PR[90,1] + 3.301;
   1:  PR[91,2] = PR[90,2] + 13.152;
   1:  PR[91,3] = PR[90,3] + 21.908;
   1:L PR[91] R[100]mm/sec CNT100;
   1:  PR[91,1] = PR[90,1] + 2.610;
   1:  PR[91,2] = PR[90,2] + 12.501;
   1:  PR[91,3] = PR[90,3] + 21.915;
   1:L PR[91] R[100]mm/sec CNT100;
   1:  PR[91,1] = PR[90,1] + 1.785;
   1:  PR[91,2] = PR[90,2] + 11.652;
   1:  PR[91,3] = PR[90,3] + 21.921;
   1:L PR[91] R[100]mm/sec CNT100;
   1:  PR[91,1] = PR[90,1] + 1.365;
   1:  PR[91,2] = PR[90,2] + 11.347;
   1:  PR[91,3] = PR[90,3] + 21.930;
   1:L PR[91] R[100]mm/sec CNT100;
   1:  PR[91,1] = PR[90,1] + 0.906;
   1:  PR[91,2] = PR[90,2] + 11.122;
   1:  PR[91,3] = PR[90,3] + 21.934;
   1:L PR[91] R[100]mm/sec CNT100;
   1:  PR[91,1] = PR[90,1] + 0.421;
   1:  PR[91,2] = PR[90,2] + 10.983;
   1:  PR[91,3] = PR[90,3] + 21.937;
   1:L PR[91] R[100]mm/sec CNT100;
   1:  PR[91,1] = PR[90,1] + -0.074;
   1:  PR[91,2] = PR[90,2] + 10.933;
   1:  PR[91,3] = PR[90,3] + 21.941;
   1:L PR[91] R[100]mm/sec CNT100;
   1:  PR[91,1] = PR[90,1] + -0.572;
   1:  PR[91,2] = PR[90,2] + 10.968;
   1:  PR[91,3] = PR[90,3] + 21.944;
   1:L PR[91] R[100]mm/sec CNT100;
   1:  PR[91,1] = PR[90,1] + -1.057;
   1:  PR[91,2] = PR[90,2] + 11.096;
   1:  PR[91,3] = PR[90,3] + 21.948;
   1:L PR[91] R[100]mm/sec CNT100;
   1:  PR[91,1] = PR[90,1] + -1.504;
   1:  PR[91,2] = PR[90,2] + 11.296;
   1:  PR[91,3] = PR[90,3] + 21.952;
   1:L PR[91] R[100]mm/sec CNT100;
   1:  PR[91,1] = PR[90,1] + -1.920;
   1:  PR[91,2] = PR[90,2] + 11.573;
   1:  PR[91,3] = PR[90,3] + 21.955;
   1:L PR[91] R[100]mm/sec CNT100;
   1:  PR[91,1] = PR[90,1] + -2.264;
   1:  PR[91,2] = PR[90,2] + 11.897;
   1:  PR[91,3] = PR[90,3] + 21.959;
   1:L PR[91] R[100]mm/sec CNT100;
   1:  PR[91,1] = PR[90,1] + -2.858;
   1:  PR[91,2] = PR[90,2] + 12.513;
   1:  PR[91,3] = PR[90,3] + 21.962;
   1:L PR[91] R[100]mm/sec CNT100;
   1:  PR[91,1] = PR[90,1] + -3.557;
   1:  PR[91,2] = PR[90,2] + 13.167;
   1:  PR[91,3] = PR[90,3] + 21.968;
   1:L PR[91] R[100]mm/sec CNT100;
   1:  PR[91,1] = PR[90,1] + -4.287;
   1:  PR[91,2] = PR[90,2] + 13.782;
   1:  PR[91,3] = PR[90,3] + 21.975;
   1:L PR[91] R[100]mm/sec CNT100;
   1:  PR[91,1] = PR[90,1] + -5.018;
   1:  PR[91,2] = PR[90,2] + 14.336;
   1:  PR[91,3] = PR[90,3] + 21.982;
   1:L PR[91] R[100]mm/sec CNT100;
   1:  PR[91,1] = PR[90,1] + -5.862;
   1:  PR[91,2] = PR[90,2] + 14.908;
   1:  PR[91,3] = PR[90,3] + 21.988;
   1:L PR[91] R[100]mm/sec CNT100;
   1:  PR[91,1] = PR[90,1] + -6.615;
   1:  PR[91,2] = PR[90,2] + 15.364;
   1:  PR[91,3] = PR[90,3] + 21.995;
   1:L PR[91] R[100]mm/sec CNT100;
   1:  PR[91,1] = PR[90,1] + -7.559;
   1:  PR[91,2] = PR[90,2] + 15.873;
   1:  PR[91,3] = PR[90,3] + 22.002;
   1:L PR[91] R[100]mm/sec CNT100;
   1:  PR[91,1] = PR[90,1] + -8.316;
   1:  PR[91,2] = PR[90,2] + 16.233;
   1:  PR[91,3] = PR[90,3] + 22.009;
   1:L PR[91] R[100]mm/sec CNT100;
   1:  PR[91,1] = PR[90,1] + -9.354;
   1:  PR[91,2] = PR[90,2] + 16.664;
   1:  PR[91,3] = PR[90,3] + 22.015;
   1:L PR[91] R[100]mm/sec CNT100;
   1:  PR[91,1] = PR[90,1] + -10.098;
   1:  PR[91,2] = PR[90,2] + 16.931;
   1:  PR[91,3] = PR[90,3] + 22.023;
   1:L PR[91] R[100]mm/sec CNT100;
   1:  PR[91,1] = PR[90,1] + -11.224;
   1:  PR[91,2] = PR[90,2] + 17.271;
   1:  PR[91,3] = PR[90,3] + 22.029;
   1:L PR[91] R[100]mm/sec CNT100;
   1:  PR[91,1] = PR[90,1] + -11.942;
   1:  PR[91,2] = PR[90,2] + 17.450;
   1:  PR[91,3] = PR[90,3] + 22.037;
   1:L PR[91] R[100]mm/sec CNT100;
   1:  PR[91,1] = PR[90,1] + -12.421;
   1:  PR[91,2] = PR[90,2] + 17.552;
   1:  PR[91,3] = PR[90,3] + 22.043;
   1:L PR[91] R[100]mm/sec CNT100;
   1:  PR[91,1] = PR[90,1] + -13.139;
   1:  PR[91,2] = PR[90,2] + 17.685;
   1:  PR[91,3] = PR[90,3] + 22.046;
   1:L PR[91] R[100]mm/sec CNT100;
   1:  PR[91,1] = PR[90,1] + -13.813;
   1:  PR[91,2] = PR[90,2] + 17.784;
   1:  PR[91,3] = PR[90,3] + 22.051;
   1:L PR[91] R[100]mm/sec CNT100;
   1:  PR[91,1] = PR[90,1] + -15.084;
   1:  PR[91,2] = PR[90,2] + 17.908;
   1:  PR[91,3] = PR[90,3] + 22.056;
   1:L PR[91] R[100]mm/sec CNT100;
   1:  PR[91,1] = PR[90,1] + -16.249;
   1:  PR[91,2] = PR[90,2] + 17.951;
   1:  PR[91,3] = PR[90,3] + 22.065;
   1:L PR[91] R[100]mm/sec CNT100;
   1:  PR[91,1] = PR[90,1] + -16.954;
   1:  PR[91,2] = PR[90,2] + 17.946;
   1:  PR[91,3] = PR[90,3] + 22.074;
   1:L PR[91] R[100]mm/sec CNT100;
   1:  PR[91,1] = PR[90,1] + -17.747;
   1:  PR[91,2] = PR[90,2] + 17.909;
   1:  PR[91,3] = PR[90,3] + 22.079;
   1:L PR[91] R[100]mm/sec CNT100;
   1:  PR[91,1] = PR[90,1] + -18.736;
   1:  PR[91,2] = PR[90,2] + 17.818;
   1:  PR[91,3] = PR[90,3] + 22.084;
   1:L PR[91] R[100]mm/sec CNT100;
   1:  PR[91,1] = PR[90,1] + -19.610;
   1:  PR[91,2] = PR[90,2] + 17.696;
   1:  PR[91,3] = PR[90,3] + 22.091;
   1:L PR[91] R[100]mm/sec CNT100;
   1:  PR[91,1] = PR[90,1] + -20.525;
   1:  PR[91,2] = PR[90,2] + 17.525;
   1:  PR[91,3] = PR[90,3] + 22.098;
   1:L PR[91] R[100]mm/sec CNT100;
   1:  PR[91,1] = PR[90,1] + -21.427;
   1:  PR[91,2] = PR[90,2] + 17.312;
   1:  PR[91,3] = PR[90,3] + 22.104;
   1:L PR[91] R[100]mm/sec CNT100;
   1:  PR[91,1] = PR[90,1] + -22.314;
   1:  PR[91,2] = PR[90,2] + 17.058;
   1:  PR[91,3] = PR[90,3] + 22.111;
   1:L PR[91] R[100]mm/sec CNT100;
   1:  PR[91,1] = PR[90,1] + -22.613;
   1:  PR[91,2] = PR[90,2] + 16.958;
   1:  PR[91,3] = PR[90,3] + 22.118;
   1:L PR[91] R[100]mm/sec CNT100;
   1:  PR[91,1] = PR[90,1] + -23.180;
   1:  PR[91,2] = PR[90,2] + 16.764;
   1:  PR[91,3] = PR[90,3] + 22.120;
   1:L PR[91] R[100]mm/sec CNT100;
   1:  PR[91,1] = PR[90,1] + -24.029;
   1:  PR[91,2] = PR[90,2] + 16.430;
   1:  PR[91,3] = PR[90,3] + 22.124;
   1:L PR[91] R[100]mm/sec CNT100;
   1:  PR[91,1] = PR[90,1] + -24.831;
   1:  PR[91,2] = PR[90,2] + 16.070;
   1:  PR[91,3] = PR[90,3] + 22.131;
   1:L PR[91] R[100]mm/sec CNT100;
   1:  PR[91,1] = PR[90,1] + -25.588;
   1:  PR[91,2] = PR[90,2] + 15.688;
   1:  PR[91,3] = PR[90,3] + 22.137;
   1:L PR[91] R[100]mm/sec CNT100;
   1:  PR[91,1] = PR[90,1] + -26.329;
   1:  PR[91,2] = PR[90,2] + 15.271;
   1:  PR[91,3] = PR[90,3] + 22.143;
   1:L PR[91] R[100]mm/sec CNT100;
   1:  PR[91,1] = PR[90,1] + -27.052;
   1:  PR[91,2] = PR[90,2] + 14.821;
   1:  PR[91,3] = PR[90,3] + 22.149;
   1:L PR[91] R[100]mm/sec CNT100;
   1:  PR[91,1] = PR[90,1] + -27.755;
   1:  PR[91,2] = PR[90,2] + 14.336;
   1:  PR[91,3] = PR[90,3] + 22.155;
   1:L PR[91] R[100]mm/sec CNT100;
   1:  PR[91,1] = PR[90,1] + -28.198;
   1:  PR[91,2] = PR[90,2] + 14.003;
   1:  PR[91,3] = PR[90,3] + 22.161;
   1:L PR[91] R[100]mm/sec CNT100;
   1:  PR[91,1] = PR[90,1] + -29.093;
   1:  PR[91,2] = PR[90,2] + 13.271;
   1:  PR[91,3] = PR[90,3] + 22.165;
   1:L PR[91] R[100]mm/sec CNT100;
   1:  PR[91,1] = PR[90,1] + -29.720;
   1:  PR[91,2] = PR[90,2] + 12.694;
   1:  PR[91,3] = PR[90,3] + 22.173;
   1:L PR[91] R[100]mm/sec CNT100;
   1:  PR[91,1] = PR[90,1] + -30.322;
   1:  PR[91,2] = PR[90,2] + 12.084;
   1:  PR[91,3] = PR[90,3] + 22.179;
   1:L PR[91] R[100]mm/sec CNT100;
   1:  PR[91,1] = PR[90,1] + -30.904;
   1:  PR[91,2] = PR[90,2] + 11.430;
   1:  PR[91,3] = PR[90,3] + 22.186;
   1:L PR[91] R[100]mm/sec CNT100;
   1:  PR[91,1] = PR[90,1] + -31.451;
   1:  PR[91,2] = PR[90,2] + 10.749;
   1:  PR[91,3] = PR[90,3] + 22.192;
   1:L PR[91] R[100]mm/sec CNT100;
   1:  PR[91,1] = PR[90,1] + -31.962;
   1:  PR[91,2] = PR[90,2] + 10.042;
   1:  PR[91,3] = PR[90,3] + 22.198;
   1:L PR[91] R[100]mm/sec CNT100;
   1:  PR[91,1] = PR[90,1] + -32.435;
   1:  PR[91,2] = PR[90,2] + 9.311;
   1:  PR[91,3] = PR[90,3] + 22.204;
   1:L PR[91] R[100]mm/sec CNT100;
   1:  PR[91,1] = PR[90,1] + -32.871;
   1:  PR[91,2] = PR[90,2] + 8.561;
   1:  PR[91,3] = PR[90,3] + 22.210;
   1:L PR[91] R[100]mm/sec CNT100;
   1:  PR[91,1] = PR[90,1] + -33.268;
   1:  PR[91,2] = PR[90,2] + 7.794;
   1:  PR[91,3] = PR[90,3] + 22.217;
   1:L PR[91] R[100]mm/sec CNT100;
   1:  PR[91,1] = PR[90,1] + -33.625;
   1:  PR[91,2] = PR[90,2] + 7.015;
   1:  PR[91,3] = PR[90,3] + 22.223;
   1:L PR[91] R[100]mm/sec CNT100;
   1:  PR[91,1] = PR[90,1] + -33.942;
   1:  PR[91,2] = PR[90,2] + 6.230;
   1:  PR[91,3] = PR[90,3] + 22.229;
   1:L PR[91] R[100]mm/sec CNT100;
   1:  PR[91,1] = PR[90,1] + -34.217;
   1:  PR[91,2] = PR[90,2] + 5.440;
   1:  PR[91,3] = PR[90,3] + 22.235;
   1:L PR[91] R[100]mm/sec CNT100;
   1:  PR[91,1] = PR[90,1] + -34.451;
   1:  PR[91,2] = PR[90,2] + 4.645;
   1:  PR[91,3] = PR[90,3] + 22.241;
   1:L PR[91] R[100]mm/sec CNT100;
   1:  PR[91,1] = PR[90,1] + -34.642;
   1:  PR[91,2] = PR[90,2] + 3.841;
   1:  PR[91,3] = PR[90,3] + 22.247;
   1:L PR[91] R[100]mm/sec CNT100;
   1:  PR[91,1] = PR[90,1] + -34.791;
   1:  PR[91,2] = PR[90,2] + 3.024;
   1:  PR[91,3] = PR[90,3] + 22.253;
   1:L PR[91] R[100]mm/sec CNT100;
   1:  PR[91,1] = PR[90,1] + -34.898;
   1:  PR[91,2] = PR[90,2] + 2.187;
   1:  PR[91,3] = PR[90,3] + 22.259;
   1:L PR[91] R[100]mm/sec CNT100;
   1:  PR[91,1] = PR[90,1] + -34.962;
   1:  PR[91,2] = PR[90,2] + 1.323;
   1:  PR[91,3] = PR[90,3] + 22.265;
   1:L PR[91] R[100]mm/sec CNT100;
   1:  PR[91,1] = PR[90,1] + -34.984;
   1:  PR[91,2] = PR[90,2] + 0.428;
   1:  PR[91,3] = PR[90,3] + 22.271;
   1:L PR[91] R[100]mm/sec CNT100;
   1:  PR[91,1] = PR[90,1] + -34.962;
   1:  PR[91,2] = PR[90,2] + -0.468;
   1:  PR[91,3] = PR[90,3] + 22.277;
   1:L PR[91] R[100]mm/sec CNT100;
   1:  PR[91,1] = PR[90,1] + -34.898;
   1:  PR[91,2] = PR[90,2] + -1.332;
   1:  PR[91,3] = PR[90,3] + 22.284;
   1:L PR[91] R[100]mm/sec CNT100;
   1:  PR[91,1] = PR[90,1] + -34.791;
   1:  PR[91,2] = PR[90,2] + -2.169;
   1:  PR[91,3] = PR[90,3] + 22.290;
   1:L PR[91] R[100]mm/sec CNT100;
   1:  PR[91,1] = PR[90,1] + -34.642;
   1:  PR[91,2] = PR[90,2] + -2.986;
   1:  PR[91,3] = PR[90,3] + 22.296;
   1:L PR[91] R[100]mm/sec CNT100;
   1:  PR[91,1] = PR[90,1] + -34.451;
   1:  PR[91,2] = PR[90,2] + -3.789;
   1:  PR[91,3] = PR[90,3] + 22.302;
   1:L PR[91] R[100]mm/sec CNT100;
   1:  PR[91,1] = PR[90,1] + -34.217;
   1:  PR[91,2] = PR[90,2] + -4.585;
   1:  PR[91,3] = PR[90,3] + 22.308;
   1:L PR[91] R[100]mm/sec CNT100;
   1:  PR[91,1] = PR[90,1] + -33.942;
   1:  PR[91,2] = PR[90,2] + -5.375;
   1:  PR[91,3] = PR[90,3] + 22.314;
   1:L PR[91] R[100]mm/sec CNT100;
   1:  PR[91,1] = PR[90,1] + -33.625;
   1:  PR[91,2] = PR[90,2] + -6.160;
   1:  PR[91,3] = PR[90,3] + 22.319;
   1:L PR[91] R[100]mm/sec CNT100;
   1:  PR[91,1] = PR[90,1] + -33.268;
   1:  PR[91,2] = PR[90,2] + -6.939;
   1:  PR[91,3] = PR[90,3] + 22.326;
   1:L PR[91] R[100]mm/sec CNT100;
   1:  PR[91,1] = PR[90,1] + -32.871;
   1:  PR[91,2] = PR[90,2] + -7.706;
   1:  PR[91,3] = PR[90,3] + 22.332;
   1:L PR[91] R[100]mm/sec CNT100;
   1:  PR[91,1] = PR[90,1] + -32.435;
   1:  PR[91,2] = PR[90,2] + -8.456;
   1:  PR[91,3] = PR[90,3] + 22.338;
   1:L PR[91] R[100]mm/sec CNT100;
   1:  PR[91,1] = PR[90,1] + -31.962;
   1:  PR[91,2] = PR[90,2] + -9.187;
   1:  PR[91,3] = PR[90,3] + 22.344;
   1:L PR[91] R[100]mm/sec CNT100;
   1:  PR[91,1] = PR[90,1] + -31.451;
   1:  PR[91,2] = PR[90,2] + -9.894;
   1:  PR[91,3] = PR[90,3] + 22.350;
   1:L PR[91] R[100]mm/sec CNT100;
   1:  PR[91,1] = PR[90,1] + -30.904;
   1:  PR[91,2] = PR[90,2] + -10.575;
   1:  PR[91,3] = PR[90,3] + 22.356;
   1:L PR[91] R[100]mm/sec CNT100;
   1:  PR[91,1] = PR[90,1] + -30.320;
   1:  PR[91,2] = PR[90,2] + -11.232;
   1:  PR[91,3] = PR[90,3] + 22.363;
   1:L PR[91] R[100]mm/sec CNT100;
   1:  PR[91,1] = PR[90,1] + -29.720;
   1:  PR[91,2] = PR[90,2] + -11.839;
   1:  PR[91,3] = PR[90,3] + 22.369;
   1:L PR[91] R[100]mm/sec CNT100;
   1:  PR[91,1] = PR[90,1] + -29.091;
   1:  PR[91,2] = PR[90,2] + -12.418;
   1:  PR[91,3] = PR[90,3] + 22.375;
   1:L PR[91] R[100]mm/sec CNT100;
   1:  PR[91,1] = PR[90,1] + -28.434;
   1:  PR[91,2] = PR[90,2] + -12.966;
   1:  PR[91,3] = PR[90,3] + 22.381;
   1:L PR[91] R[100]mm/sec CNT100;
   1:  PR[91,1] = PR[90,1] + -27.754;
   1:  PR[91,2] = PR[90,2] + -13.482;
   1:  PR[91,3] = PR[90,3] + 22.387;
   1:L PR[91] R[100]mm/sec CNT100;
   1:  PR[91,1] = PR[90,1] + -27.051;
   1:  PR[91,2] = PR[90,2] + -13.966;
   1:  PR[91,3] = PR[90,3] + 22.393;
   1:L PR[91] R[100]mm/sec CNT100;
   1:  PR[91,1] = PR[90,1] + -26.613;
   1:  PR[91,2] = PR[90,2] + -14.242;
   1:  PR[91,3] = PR[90,3] + 22.399;
   1:L PR[91] R[100]mm/sec CNT100;
   1:  PR[91,1] = PR[90,1] + -25.585;
   1:  PR[91,2] = PR[90,2] + -14.834;
   1:  PR[91,3] = PR[90,3] + 22.403;
   1:L PR[91] R[100]mm/sec CNT100;
   1:  PR[91,1] = PR[90,1] + -24.831;
   1:  PR[91,2] = PR[90,2] + -15.215;
   1:  PR[91,3] = PR[90,3] + 22.411;
   1:L PR[91] R[100]mm/sec CNT100;
   1:  PR[91,1] = PR[90,1] + -24.029;
   1:  PR[91,2] = PR[90,2] + -15.575;
   1:  PR[91,3] = PR[90,3] + 22.418;
   1:L PR[91] R[100]mm/sec CNT100;
   1:  PR[91,1] = PR[90,1] + -23.180;
   1:  PR[91,2] = PR[90,2] + -15.909;
   1:  PR[91,3] = PR[90,3] + 22.424;
   1:L PR[91] R[100]mm/sec CNT100;
   1:  PR[91,1] = PR[90,1] + -22.613;
   1:  PR[91,2] = PR[90,2] + -16.103;
   1:  PR[91,3] = PR[90,3] + 22.430;
   1:L PR[91] R[100]mm/sec CNT100;
   1:  PR[91,1] = PR[90,1] + -22.314;
   1:  PR[91,2] = PR[90,2] + -16.203;
   1:  PR[91,3] = PR[90,3] + 22.435;
   1:L PR[91] R[100]mm/sec CNT100;
   1:  PR[91,1] = PR[90,1] + -21.427;
   1:  PR[91,2] = PR[90,2] + -16.457;
   1:  PR[91,3] = PR[90,3] + 22.437;
   1:L PR[91] R[100]mm/sec CNT100;
   1:  PR[91,1] = PR[90,1] + -20.526;
   1:  PR[91,2] = PR[90,2] + -16.670;
   1:  PR[91,3] = PR[90,3] + 22.443;
   1:L PR[91] R[100]mm/sec CNT100;
   1:  PR[91,1] = PR[90,1] + -19.610;
   1:  PR[91,2] = PR[90,2] + -16.841;
   1:  PR[91,3] = PR[90,3] + 22.450;
   1:L PR[91] R[100]mm/sec CNT100;
   1:  PR[91,1] = PR[90,1] + -18.735;
   1:  PR[91,2] = PR[90,2] + -16.962;
   1:  PR[91,3] = PR[90,3] + 22.457;
   1:L PR[91] R[100]mm/sec CNT100;
   1:  PR[91,1] = PR[90,1] + -17.951;
   1:  PR[91,2] = PR[90,2] + -17.037;
   1:  PR[91,3] = PR[90,3] + 22.463;
   1:L PR[91] R[100]mm/sec CNT100;
   1:  PR[91,1] = PR[90,1] + -16.955;
   1:  PR[91,2] = PR[90,2] + -17.090;
   1:  PR[91,3] = PR[90,3] + 22.469;
   1:L PR[91] R[100]mm/sec CNT100;
   1:  PR[91,1] = PR[90,1] + -15.776;
   1:  PR[91,2] = PR[90,2] + -17.087;
   1:  PR[91,3] = PR[90,3] + 22.476;
   1:L PR[91] R[100]mm/sec CNT100;
   1:  PR[91,1] = PR[90,1] + -15.084;
   1:  PR[91,2] = PR[90,2] + -17.053;
   1:  PR[91,3] = PR[90,3] + 22.484;
   1:L PR[91] R[100]mm/sec CNT100;
   1:  PR[91,1] = PR[90,1] + -14.422;
   1:  PR[91,2] = PR[90,2] + -16.998;
   1:  PR[91,3] = PR[90,3] + 22.489;
   1:L PR[91] R[100]mm/sec CNT100;
   1:  PR[91,1] = PR[90,1] + -13.818;
   1:  PR[91,2] = PR[90,2] + -16.930;
   1:  PR[91,3] = PR[90,3] + 22.494;
   1:L PR[91] R[100]mm/sec CNT100;
   1:  PR[91,1] = PR[90,1] + -13.142;
   1:  PR[91,2] = PR[90,2] + -16.830;
   1:  PR[91,3] = PR[90,3] + 22.498;
   1:L PR[91] R[100]mm/sec CNT100;
   1:  PR[91,1] = PR[90,1] + -11.937;
   1:  PR[91,2] = PR[90,2] + -16.593;
   1:  PR[91,3] = PR[90,3] + 22.503;
   1:L PR[91] R[100]mm/sec CNT100;
   1:  PR[91,1] = PR[90,1] + -11.222;
   1:  PR[91,2] = PR[90,2] + -16.415;
   1:  PR[91,3] = PR[90,3] + 22.512;
   1:L PR[91] R[100]mm/sec CNT100;
   1:  PR[91,1] = PR[90,1] + -10.471;
   1:  PR[91,2] = PR[90,2] + -16.196;
   1:  PR[91,3] = PR[90,3] + 22.517;
   1:L PR[91] R[100]mm/sec CNT100;
   1:  PR[91,1] = PR[90,1] + -9.352;
   1:  PR[91,2] = PR[90,2] + -15.808;
   1:  PR[91,3] = PR[90,3] + 22.523;
   1:L PR[91] R[100]mm/sec CNT100;
   1:  PR[91,1] = PR[90,1] + -8.316;
   1:  PR[91,2] = PR[90,2] + -15.378;
   1:  PR[91,3] = PR[90,3] + 22.531;
   1:L PR[91] R[100]mm/sec CNT100;
   1:  PR[91,1] = PR[90,1] + -7.559;
   1:  PR[91,2] = PR[90,2] + -15.018;
   1:  PR[91,3] = PR[90,3] + 22.539;
   1:L PR[91] R[100]mm/sec CNT100;
   1:  PR[91,1] = PR[90,1] + -6.616;
   1:  PR[91,2] = PR[90,2] + -14.510;
   1:  PR[91,3] = PR[90,3] + 22.545;
   1:L PR[91] R[100]mm/sec CNT100;
   1:  PR[91,1] = PR[90,1] + -5.862;
   1:  PR[91,2] = PR[90,2] + -14.053;
   1:  PR[91,3] = PR[90,3] + 22.553;
   1:L PR[91] R[100]mm/sec CNT100;
   1:  PR[91,1] = PR[90,1] + -5.100;
   1:  PR[91,2] = PR[90,2] + -13.538;
   1:  PR[91,3] = PR[90,3] + 22.559;
   1:L PR[91] R[100]mm/sec CNT100;
   1:  PR[91,1] = PR[90,1] + -4.288;
   1:  PR[91,2] = PR[90,2] + -12.927;
   1:  PR[91,3] = PR[90,3] + 22.565;
   1:L PR[91] R[100]mm/sec CNT100;
   1:  PR[91,1] = PR[90,1] + -3.531;
   1:  PR[91,2] = PR[90,2] + -12.288;
   1:  PR[91,3] = PR[90,3] + 22.573;
   1:L PR[91] R[100]mm/sec CNT100;
   1:  PR[91,1] = PR[90,1] + -2.858;
   1:  PR[91,2] = PR[90,2] + -11.658;
   1:  PR[91,3] = PR[90,3] + 22.580;
   1:L PR[91] R[100]mm/sec CNT100;
   1:  PR[91,1] = PR[90,1] + -2.264;
   1:  PR[91,2] = PR[90,2] + -11.040;
   1:  PR[91,3] = PR[90,3] + 22.586;
   1:L PR[91] R[100]mm/sec CNT100;
   1:  PR[91,1] = PR[90,1] + -1.919;
   1:  PR[91,2] = PR[90,2] + -10.717;
   1:  PR[91,3] = PR[90,3] + 22.592;
   1:L PR[91] R[100]mm/sec CNT100;
   1:  PR[91,1] = PR[90,1] + -1.503;
   1:  PR[91,2] = PR[90,2] + -10.440;
   1:  PR[91,3] = PR[90,3] + 22.596;
   1:L PR[91] R[100]mm/sec CNT100;
   1:  PR[91,1] = PR[90,1] + -1.048;
   1:  PR[91,2] = PR[90,2] + -10.238;
   1:  PR[91,3] = PR[90,3] + 22.599;
   1:L PR[91] R[100]mm/sec CNT100;
   1:  PR[91,1] = PR[90,1] + -0.572;
   1:  PR[91,2] = PR[90,2] + -10.113;
   1:  PR[91,3] = PR[90,3] + 22.603;
   1:L PR[91] R[100]mm/sec CNT100;
   1:  PR[91,1] = PR[90,1] + -0.074;
   1:  PR[91,2] = PR[90,2] + -10.078;
   1:  PR[91,3] = PR[90,3] + 22.606;
   1:L PR[91] R[100]mm/sec CNT100;
   1:  PR[91] = PR[90];
   1:  PR[91,1] = PR[90,1] + 0.538;
   1:  PR[91,2] = PR[90,2] + -10.869;
   1:  PR[91,3] = PR[90,3] + 23.940;
   1:L PR[91] R[100]mm/sec CNT100;
   1:  PR[91,1] = PR[90,1] + 1.013;
   1:  PR[91,2] = PR[90,2] + -11.027;
   1:  PR[91,3] = PR[90,3] + 22.614;
   1:L PR[91] R[100]mm/sec CNT100;
   1:  PR[91,1] = PR[90,1] + 1.461;
   1:  PR[91,2] = PR[90,2] + -11.264;
   1:  PR[91,3] = PR[90,3] + 22.617;
   1:L PR[91] R[100]mm/sec CNT100;
   1:  PR[91,1] = PR[90,1] + 1.855;
   1:  PR[91,2] = PR[90,2] + -11.569;
   1:  PR[91,3] = PR[90,3] + 22.621;
   1:L PR[91] R[100]mm/sec CNT100;
   1:  PR[91,1] = PR[90,1] + 2.684;
   1:  PR[91,2] = PR[90,2] + -12.365;
   1:  PR[91,3] = PR[90,3] + 22.624;
   1:L PR[91] R[100]mm/sec CNT100;
   1:  PR[91,1] = PR[90,1] + 3.419;
   1:  PR[91,2] = PR[90,2] + -12.988;
   1:  PR[91,3] = PR[90,3] + 22.633;
   1:L PR[91] R[100]mm/sec CNT100;
   1:  PR[91,1] = PR[90,1] + 3.676;
   1:  PR[91,2] = PR[90,2] + -13.186;
   1:  PR[91,3] = PR[90,3] + 22.640;
   1:L PR[91] R[100]mm/sec CNT100;
   1:  PR[91,1] = PR[90,1] + 4.186;
   1:  PR[91,2] = PR[90,2] + -13.571;
   1:  PR[91,3] = PR[90,3] + 22.642;
   1:L PR[91] R[100]mm/sec CNT100;
   1:  PR[91,1] = PR[90,1] + 4.992;
   1:  PR[91,2] = PR[90,2] + -14.118;
   1:  PR[91,3] = PR[90,3] + 22.647;
   1:L PR[91] R[100]mm/sec CNT100;
   1:  PR[91,1] = PR[90,1] + 5.828;
   1:  PR[91,2] = PR[90,2] + -14.624;
   1:  PR[91,3] = PR[90,3] + 22.654;
   1:L PR[91] R[100]mm/sec CNT100;
   1:  PR[91,1] = PR[90,1] + 6.695;
   1:  PR[91,2] = PR[90,2] + -15.089;
   1:  PR[91,3] = PR[90,3] + 22.661;
   1:L PR[91] R[100]mm/sec CNT100;
   1:  PR[91,1] = PR[90,1] + 7.590;
   1:  PR[91,2] = PR[90,2] + -15.511;
   1:  PR[91,3] = PR[90,3] + 22.668;
   1:L PR[91] R[100]mm/sec CNT100;
   1:  PR[91,1] = PR[90,1] + 8.505;
   1:  PR[91,2] = PR[90,2] + -15.888;
   1:  PR[91,3] = PR[90,3] + 22.675;
   1:L PR[91] R[100]mm/sec CNT100;
   1:  PR[91,1] = PR[90,1] + 9.399;
   1:  PR[91,2] = PR[90,2] + -16.207;
   1:  PR[91,3] = PR[90,3] + 22.682;
   1:L PR[91] R[100]mm/sec CNT100;
   1:  PR[91,1] = PR[90,1] + 10.381;
   1:  PR[91,2] = PR[90,2] + -16.503;
   1:  PR[91,3] = PR[90,3] + 22.689;
   1:L PR[91] R[100]mm/sec CNT100;
   1:  PR[91,1] = PR[90,1] + 11.434;
   1:  PR[91,2] = PR[90,2] + -16.759;
   1:  PR[91,3] = PR[90,3] + 22.696;
   1:L PR[91] R[100]mm/sec CNT100;
   1:  PR[91,1] = PR[90,1] + 12.311;
   1:  PR[91,2] = PR[90,2] + -16.928;
   1:  PR[91,3] = PR[90,3] + 22.704;
   1:L PR[91] R[100]mm/sec CNT100;
   1:  PR[91,1] = PR[90,1] + 13.147;
   1:  PR[91,2] = PR[90,2] + -17.050;
   1:  PR[91,3] = PR[90,3] + 22.711;
   1:L PR[91] R[100]mm/sec CNT100;
   1:  PR[91,1] = PR[90,1] + 13.939;
   1:  PR[91,2] = PR[90,2] + -17.130;
   1:  PR[91,3] = PR[90,3] + 22.717;
   1:L PR[91] R[100]mm/sec CNT100;
   1:  PR[91,1] = PR[90,1] + 15.055;
   1:  PR[91,2] = PR[90,2] + -17.194;
   1:  PR[91,3] = PR[90,3] + 22.723;
   1:L PR[91] R[100]mm/sec CNT100;
   1:  PR[91,1] = PR[90,1] + 16.236;
   1:  PR[91,2] = PR[90,2] + -17.193;
   1:  PR[91,3] = PR[90,3] + 22.731;
   1:L PR[91] R[100]mm/sec CNT100;
   1:  PR[91,1] = PR[90,1] + 16.955;
   1:  PR[91,2] = PR[90,2] + -17.157;
   1:  PR[91,3] = PR[90,3] + 22.739;
   1:L PR[91] R[100]mm/sec CNT100;
   1:  PR[91,1] = PR[90,1] + 18.186;
   1:  PR[91,2] = PR[90,2] + -17.037;
   1:  PR[91,3] = PR[90,3] + 22.744;
   1:L PR[91] R[100]mm/sec CNT100;
   1:  PR[91,1] = PR[90,1] + 18.837;
   1:  PR[91,2] = PR[90,2] + -16.942;
   1:  PR[91,3] = PR[90,3] + 22.753;
   1:L PR[91] R[100]mm/sec CNT100;
   1:  PR[91,1] = PR[90,1] + 20.050;
   1:  PR[91,2] = PR[90,2] + -16.707;
   1:  PR[91,3] = PR[90,3] + 22.758;
   1:L PR[91] R[100]mm/sec CNT100;
   1:  PR[91,1] = PR[90,1] + 20.700;
   1:  PR[91,2] = PR[90,2] + -16.549;
   1:  PR[91,3] = PR[90,3] + 22.767;
   1:L PR[91] R[100]mm/sec CNT100;
   1:  PR[91,1] = PR[90,1] + 21.745;
   1:  PR[91,2] = PR[90,2] + -16.243;
   1:  PR[91,3] = PR[90,3] + 22.772;
   1:L PR[91] R[100]mm/sec CNT100;
   1:  PR[91,1] = PR[90,1] + 22.457;
   1:  PR[91,2] = PR[90,2] + -16.001;
   1:  PR[91,3] = PR[90,3] + 22.780;
   1:L PR[91] R[100]mm/sec CNT100;
   1:  PR[91,1] = PR[90,1] + 23.231;
   1:  PR[91,2] = PR[90,2] + -15.701;
   1:  PR[91,3] = PR[90,3] + 22.785;
   1:L PR[91] R[100]mm/sec CNT100;
   1:  PR[91,1] = PR[90,1] + 24.081;
   1:  PR[91,2] = PR[90,2] + -15.328;
   1:  PR[91,3] = PR[90,3] + 22.791;
   1:L PR[91] R[100]mm/sec CNT100;
   1:  PR[91,1] = PR[90,1] + 24.891;
   1:  PR[91,2] = PR[90,2] + -14.925;
   1:  PR[91,3] = PR[90,3] + 22.798;
   1:L PR[91] R[100]mm/sec CNT100;
   1:  PR[91,1] = PR[90,1] + 25.683;
   1:  PR[91,2] = PR[90,2] + -14.483;
   1:  PR[91,3] = PR[90,3] + 22.804;
   1:L PR[91] R[100]mm/sec CNT100;
   1:  PR[91,1] = PR[90,1] + 26.448;
   1:  PR[91,2] = PR[90,2] + -14.006;
   1:  PR[91,3] = PR[90,3] + 22.811;
   1:L PR[91] R[100]mm/sec CNT100;
   1:  PR[91,1] = PR[90,1] + 27.185;
   1:  PR[91,2] = PR[90,2] + -13.497;
   1:  PR[91,3] = PR[90,3] + 22.817;
   1:L PR[91] R[100]mm/sec CNT100;
   1:  PR[91,1] = PR[90,1] + 27.892;
   1:  PR[91,2] = PR[90,2] + -12.955;
   1:  PR[91,3] = PR[90,3] + 22.824;
   1:L PR[91] R[100]mm/sec CNT100;
   1:  PR[91,1] = PR[90,1] + 28.569;
   1:  PR[91,2] = PR[90,2] + -12.383;
   1:  PR[91,3] = PR[90,3] + 22.830;
   1:L PR[91] R[100]mm/sec CNT100;
   1:  PR[91,1] = PR[90,1] + 29.214;
   1:  PR[91,2] = PR[90,2] + -11.781;
   1:  PR[91,3] = PR[90,3] + 22.837;
   1:L PR[91] R[100]mm/sec CNT100;
   1:  PR[91,1] = PR[90,1] + 29.818;
   1:  PR[91,2] = PR[90,2] + -11.156;
   1:  PR[91,3] = PR[90,3] + 22.843;
   1:L PR[91] R[100]mm/sec CNT100;
   1:  PR[91,1] = PR[90,1] + 30.378;
   1:  PR[91,2] = PR[90,2] + -10.515;
   1:  PR[91,3] = PR[90,3] + 22.849;
   1:L PR[91] R[100]mm/sec CNT100;
   1:  PR[91,1] = PR[90,1] + 30.908;
   1:  PR[91,2] = PR[90,2] + -9.845;
   1:  PR[91,3] = PR[90,3] + 22.855;
   1:L PR[91] R[100]mm/sec CNT100;
   1:  PR[91,1] = PR[90,1] + 31.406;
   1:  PR[91,2] = PR[90,2] + -9.149;
   1:  PR[91,3] = PR[90,3] + 22.862;
   1:L PR[91] R[100]mm/sec CNT100;
   1:  PR[91,1] = PR[90,1] + 31.870;
   1:  PR[91,2] = PR[90,2] + -8.430;
   1:  PR[91,3] = PR[90,3] + 22.868;
   1:L PR[91] R[100]mm/sec CNT100;
   1:  PR[91,1] = PR[90,1] + 32.300;
   1:  PR[91,2] = PR[90,2] + -7.691;
   1:  PR[91,3] = PR[90,3] + 22.874;
   1:L PR[91] R[100]mm/sec CNT100;
   1:  PR[91,1] = PR[90,1] + 32.693;
   1:  PR[91,2] = PR[90,2] + -6.936;
   1:  PR[91,3] = PR[90,3] + 22.880;
   1:L PR[91] R[100]mm/sec CNT100;
   1:  PR[91,1] = PR[90,1] + 33.048;
   1:  PR[91,2] = PR[90,2] + -6.170;
   1:  PR[91,3] = PR[90,3] + 22.886;
   1:L PR[91] R[100]mm/sec CNT100;
   1:  PR[91,1] = PR[90,1] + 33.363;
   1:  PR[91,2] = PR[90,2] + -5.396;
   1:  PR[91,3] = PR[90,3] + 22.892;
   1:L PR[91] R[100]mm/sec CNT100;
   1:  PR[91,1] = PR[90,1] + 33.638;
   1:  PR[91,2] = PR[90,2] + -4.614;
   1:  PR[91,3] = PR[90,3] + 22.898;
   1:L PR[91] R[100]mm/sec CNT100;
   1:  PR[91,1] = PR[90,1] + 33.872;
   1:  PR[91,2] = PR[90,2] + -3.822;
   1:  PR[91,3] = PR[90,3] + 22.904;
   1:L PR[91] R[100]mm/sec CNT100;
   1:  PR[91,1] = PR[90,1] + 34.064;
   1:  PR[91,2] = PR[90,2] + -3.018;
   1:  PR[91,3] = PR[90,3] + 22.910;
   1:L PR[91] R[100]mm/sec CNT100;
   1:  PR[91,1] = PR[90,1] + 34.214;
   1:  PR[91,2] = PR[90,2] + -2.195;
   1:  PR[91,3] = PR[90,3] + 22.916;
   1:L PR[91] R[100]mm/sec CNT100;
   1:  PR[91,1] = PR[90,1] + 34.322;
   1:  PR[91,2] = PR[90,2] + -1.350;
   1:  PR[91,3] = PR[90,3] + 22.922;
   1:L PR[91] R[100]mm/sec CNT100;
   1:  PR[91,1] = PR[90,1] + 34.387;
   1:  PR[91,2] = PR[90,2] + -0.477;
   1:  PR[91,3] = PR[90,3] + 22.928;
   1:L PR[91] R[100]mm/sec CNT100;
   1:  PR[91,1] = PR[90,1] + 34.409;
   1:  PR[91,2] = PR[90,2] + 0.428;
   1:  PR[91,3] = PR[90,3] + 22.935;
   1:L PR[91] R[100]mm/sec CNT100;
   1:  PR[91,1] = PR[90,1] + 34.387;
   1:  PR[91,2] = PR[90,2] + 1.332;
   1:  PR[91,3] = PR[90,3] + 22.941;
   1:L PR[91] R[100]mm/sec CNT100;
   1:  PR[91,1] = PR[90,1] + 34.322;
   1:  PR[91,2] = PR[90,2] + 2.205;
   1:  PR[91,3] = PR[90,3] + 22.948;
   1:L PR[91] R[100]mm/sec CNT100;
   1:  PR[91,1] = PR[90,1] + 34.214;
   1:  PR[91,2] = PR[90,2] + 3.050;
   1:  PR[91,3] = PR[90,3] + 22.954;
   1:L PR[91] R[100]mm/sec CNT100;
   1:  PR[91,1] = PR[90,1] + 34.064;
   1:  PR[91,2] = PR[90,2] + 3.873;
   1:  PR[91,3] = PR[90,3] + 22.960;
   1:L PR[91] R[100]mm/sec CNT100;
   1:  PR[91,1] = PR[90,1] + 33.872;
   1:  PR[91,2] = PR[90,2] + 4.677;
   1:  PR[91,3] = PR[90,3] + 22.966;
   1:L PR[91] R[100]mm/sec CNT100;
   1:  PR[91,1] = PR[90,1] + 33.638;
   1:  PR[91,2] = PR[90,2] + 5.469;
   1:  PR[91,3] = PR[90,3] + 22.972;
   1:L PR[91] R[100]mm/sec CNT100;
   1:  PR[91,1] = PR[90,1] + 33.363;
   1:  PR[91,2] = PR[90,2] + 6.251;
   1:  PR[91,3] = PR[90,3] + 22.978;
   1:L PR[91] R[100]mm/sec CNT100;
   1:  PR[91,1] = PR[90,1] + 33.048;
   1:  PR[91,2] = PR[90,2] + 7.025;
   1:  PR[91,3] = PR[90,3] + 22.984;
   1:L PR[91] R[100]mm/sec CNT100;
   1:  PR[91,1] = PR[90,1] + 32.692;
   1:  PR[91,2] = PR[90,2] + 7.792;
   1:  PR[91,3] = PR[90,3] + 22.990;
   1:L PR[91] R[100]mm/sec CNT100;
   1:  PR[91,1] = PR[90,1] + 32.489;
   1:  PR[91,2] = PR[90,2] + 8.185;
   1:  PR[91,3] = PR[90,3] + 22.996;
   1:L PR[91] R[100]mm/sec CNT100;
   1:  PR[91,1] = PR[90,1] + 32.300;
   1:  PR[91,2] = PR[90,2] + 8.545;
   1:  PR[91,3] = PR[90,3] + 23.000;
   1:L PR[91] R[100]mm/sec CNT100;
   1:  PR[91,1] = PR[90,1] + 31.870;
   1:  PR[91,2] = PR[90,2] + 9.285;
   1:  PR[91,3] = PR[90,3] + 23.003;
   1:L PR[91] R[100]mm/sec CNT100;
   1:  PR[91,1] = PR[90,1] + 31.405;
   1:  PR[91,2] = PR[90,2] + 10.005;
   1:  PR[91,3] = PR[90,3] + 23.009;
   1:L PR[91] R[100]mm/sec CNT100;
   1:  PR[91,1] = PR[90,1] + 31.030;
   1:  PR[91,2] = PR[90,2] + 10.532;
   1:  PR[91,3] = PR[90,3] + 23.015;
   1:L PR[91] R[100]mm/sec CNT100;
   1:  PR[91,1] = PR[90,1] + 30.376;
   1:  PR[91,2] = PR[90,2] + 11.372;
   1:  PR[91,3] = PR[90,3] + 23.020;
   1:L PR[91] R[100]mm/sec CNT100;
   1:  PR[91,1] = PR[90,1] + 29.818;
   1:  PR[91,2] = PR[90,2] + 12.011;
   1:  PR[91,3] = PR[90,3] + 23.027;
   1:L PR[91] R[100]mm/sec CNT100;
   1:  PR[91,1] = PR[90,1] + 29.214;
   1:  PR[91,2] = PR[90,2] + 12.636;
   1:  PR[91,3] = PR[90,3] + 23.033;
   1:L PR[91] R[100]mm/sec CNT100;
   1:  PR[91,1] = PR[90,1] + 28.569;
   1:  PR[91,2] = PR[90,2] + 13.238;
   1:  PR[91,3] = PR[90,3] + 23.040;
   1:L PR[91] R[100]mm/sec CNT100;
   1:  PR[91,1] = PR[90,1] + 27.892;
   1:  PR[91,2] = PR[90,2] + 13.811;
   1:  PR[91,3] = PR[90,3] + 23.046;
   1:L PR[91] R[100]mm/sec CNT100;
   1:  PR[91,1] = PR[90,1] + 27.454;
   1:  PR[91,2] = PR[90,2] + 14.147;
   1:  PR[91,3] = PR[90,3] + 23.052;
   1:L PR[91] R[100]mm/sec CNT100;
   1:  PR[91,1] = PR[90,1] + 27.186;
   1:  PR[91,2] = PR[90,2] + 14.351;
   1:  PR[91,3] = PR[90,3] + 23.056;
   1:L PR[91] R[100]mm/sec CNT100;
   1:  PR[91,1] = PR[90,1] + 26.450;
   1:  PR[91,2] = PR[90,2] + 14.860;
   1:  PR[91,3] = PR[90,3] + 23.059;
   1:L PR[91] R[100]mm/sec CNT100;
   1:  PR[91,1] = PR[90,1] + 25.481;
   1:  PR[91,2] = PR[90,2] + 15.452;
   1:  PR[91,3] = PR[90,3] + 23.065;
   1:L PR[91] R[100]mm/sec CNT100;
   1:  PR[91,1] = PR[90,1] + 24.891;
   1:  PR[91,2] = PR[90,2] + 15.780;
   1:  PR[91,3] = PR[90,3] + 23.074;
   1:L PR[91] R[100]mm/sec CNT100;
   1:  PR[91,1] = PR[90,1] + 24.069;
   1:  PR[91,2] = PR[90,2] + 16.189;
   1:  PR[91,3] = PR[90,3] + 23.078;
   1:L PR[91] R[100]mm/sec CNT100;
   1:  PR[91,1] = PR[90,1] + 23.231;
   1:  PR[91,2] = PR[90,2] + 16.557;
   1:  PR[91,3] = PR[90,3] + 23.085;
   1:L PR[91] R[100]mm/sec CNT100;
   1:  PR[91,1] = PR[90,1] + 22.459;
   1:  PR[91,2] = PR[90,2] + 16.855;
   1:  PR[91,3] = PR[90,3] + 23.092;
   1:L PR[91] R[100]mm/sec CNT100;
   1:  PR[91,1] = PR[90,1] + 21.425;
   1:  PR[91,2] = PR[90,2] + 17.199;
   1:  PR[91,3] = PR[90,3] + 23.098;
   1:L PR[91] R[100]mm/sec CNT100;
   1:  PR[91,1] = PR[90,1] + 20.702;
   1:  PR[91,2] = PR[90,2] + 17.403;
   1:  PR[91,3] = PR[90,3] + 23.105;
   1:L PR[91] R[100]mm/sec CNT100;
   1:  PR[91,1] = PR[90,1] + 20.050;
   1:  PR[91,2] = PR[90,2] + 17.562;
   1:  PR[91,3] = PR[90,3] + 23.111;
   1:L PR[91] R[100]mm/sec CNT100;
   1:  PR[91,1] = PR[90,1] + 18.837;
   1:  PR[91,2] = PR[90,2] + 17.797;
   1:  PR[91,3] = PR[90,3] + 23.116;
   1:L PR[91] R[100]mm/sec CNT100;
   1:  PR[91,1] = PR[90,1] + 18.182;
   1:  PR[91,2] = PR[90,2] + 17.893;
   1:  PR[91,3] = PR[90,3] + 23.125;
   1:L PR[91] R[100]mm/sec CNT100;
   1:  PR[91,1] = PR[90,1] + 17.476;
   1:  PR[91,2] = PR[90,2] + 17.971;
   1:  PR[91,3] = PR[90,3] + 23.129;
   1:L PR[91] R[100]mm/sec CNT100;
   1:  PR[91,1] = PR[90,1] + 16.964;
   1:  PR[91,2] = PR[90,2] + 18.012;
   1:  PR[91,3] = PR[90,3] + 23.135;
   1:L PR[91] R[100]mm/sec CNT100;
   1:  PR[91,1] = PR[90,1] + 15.793;
   1:  PR[91,2] = PR[90,2] + 18.055;
   1:  PR[91,3] = PR[90,3] + 23.138;
   1:L PR[91] R[100]mm/sec CNT100;
   1:  PR[91,1] = PR[90,1] + 15.054;
   1:  PR[91,2] = PR[90,2] + 18.049;
   1:  PR[91,3] = PR[90,3] + 23.147;
   1:L PR[91] R[100]mm/sec CNT100;
   1:  PR[91,1] = PR[90,1] + 14.271;
   1:  PR[91,2] = PR[90,2] + 18.013;
   1:  PR[91,3] = PR[90,3] + 23.152;
   1:L PR[91] R[100]mm/sec CNT100;
   1:  PR[91,1] = PR[90,1] + 13.144;
   1:  PR[91,2] = PR[90,2] + 17.904;
   1:  PR[91,3] = PR[90,3] + 23.158;
   1:L PR[91] R[100]mm/sec CNT100;
   1:  PR[91,1] = PR[90,1] + 12.311;
   1:  PR[91,2] = PR[90,2] + 17.783;
   1:  PR[91,3] = PR[90,3] + 23.166;
   1:L PR[91] R[100]mm/sec CNT100;
   1:  PR[91,1] = PR[90,1] + 11.434;
   1:  PR[91,2] = PR[90,2] + 17.614;
   1:  PR[91,3] = PR[90,3] + 23.172;
   1:L PR[91] R[100]mm/sec CNT100;
   1:  PR[91,1] = PR[90,1] + 10.380;
   1:  PR[91,2] = PR[90,2] + 17.358;
   1:  PR[91,3] = PR[90,3] + 23.178;
   1:L PR[91] R[100]mm/sec CNT100;
   1:  PR[91,1] = PR[90,1] + 9.398;
   1:  PR[91,2] = PR[90,2] + 17.062;
   1:  PR[91,3] = PR[90,3] + 23.186;
   1:L PR[91] R[100]mm/sec CNT100;
   1:  PR[91,1] = PR[90,1] + 8.481;
   1:  PR[91,2] = PR[90,2] + 16.734;
   1:  PR[91,3] = PR[90,3] + 23.194;
   1:L PR[91] R[100]mm/sec CNT100;
   1:  PR[91,1] = PR[90,1] + 7.589;
   1:  PR[91,2] = PR[90,2] + 16.366;
   1:  PR[91,3] = PR[90,3] + 23.201;
   1:L PR[91] R[100]mm/sec CNT100;
   1:  PR[91,1] = PR[90,1] + 6.694;
   1:  PR[91,2] = PR[90,2] + 15.944;
   1:  PR[91,3] = PR[90,3] + 23.208;
   1:L PR[91] R[100]mm/sec CNT100;
   1:  PR[91,1] = PR[90,1] + 5.828;
   1:  PR[91,2] = PR[90,2] + 15.479;
   1:  PR[91,3] = PR[90,3] + 23.215;
   1:L PR[91] R[100]mm/sec CNT100;
   1:  PR[91,1] = PR[90,1] + 4.991;
   1:  PR[91,2] = PR[90,2] + 14.973;
   1:  PR[91,3] = PR[90,3] + 23.222;
   1:L PR[91] R[100]mm/sec CNT100;
   1:  PR[91,1] = PR[90,1] + 4.186;
   1:  PR[91,2] = PR[90,2] + 14.426;
   1:  PR[91,3] = PR[90,3] + 23.229;
   1:L PR[91] R[100]mm/sec CNT100;
   1:  PR[91,1] = PR[90,1] + 3.676;
   1:  PR[91,2] = PR[90,2] + 14.041;
   1:  PR[91,3] = PR[90,3] + 23.236;
   1:L PR[91] R[100]mm/sec CNT100;
   1:  PR[91,1] = PR[90,1] + 3.418;
   1:  PR[91,2] = PR[90,2] + 13.843;
   1:  PR[91,3] = PR[90,3] + 23.241;
   1:L PR[91] R[100]mm/sec CNT100;
   1:  PR[91,1] = PR[90,1] + 2.684;
   1:  PR[91,2] = PR[90,2] + 13.221;
   1:  PR[91,3] = PR[90,3] + 23.243;
   1:L PR[91] R[100]mm/sec CNT100;
   1:  PR[91,1] = PR[90,1] + 1.855;
   1:  PR[91,2] = PR[90,2] + 12.424;
   1:  PR[91,3] = PR[90,3] + 23.250;
   1:L PR[91] R[100]mm/sec CNT100;
   1:  PR[91,1] = PR[90,1] + 1.461;
   1:  PR[91,2] = PR[90,2] + 12.120;
   1:  PR[91,3] = PR[90,3] + 23.258;
   1:L PR[91] R[100]mm/sec CNT100;
   1:  PR[91,1] = PR[90,1] + 1.013;
   1:  PR[91,2] = PR[90,2] + 11.882;
   1:  PR[91,3] = PR[90,3] + 23.262;
   1:L PR[91] R[100]mm/sec CNT100;
   1:  PR[91,1] = PR[90,1] + 0.539;
   1:  PR[91,2] = PR[90,2] + 11.724;
   1:  PR[91,3] = PR[90,3] + 23.265;
   1:L PR[91] R[100]mm/sec CNT100;
   1:  PR[91,1] = PR[90,1] + 0.042;
   1:  PR[91,2] = PR[90,2] + 11.648;
   1:  PR[91,3] = PR[90,3] + 23.269;
   1:L PR[91] R[100]mm/sec CNT100;
   1:  PR[91,1] = PR[90,1] + -0.455;
   1:  PR[91,2] = PR[90,2] + 11.667;
   1:  PR[91,3] = PR[90,3] + 23.273;
   1:L PR[91] R[100]mm/sec CNT100;
   1:  PR[91,1] = PR[90,1] + -0.940;
   1:  PR[91,2] = PR[90,2] + 11.766;
   1:  PR[91,3] = PR[90,3] + 23.276;
   1:L PR[91] R[100]mm/sec CNT100;
   1:  PR[91,1] = PR[90,1] + -1.402;
   1:  PR[91,2] = PR[90,2] + 11.952;
   1:  PR[91,3] = PR[90,3] + 23.280;
   1:L PR[91] R[100]mm/sec CNT100;
   1:  PR[91,1] = PR[90,1] + -1.825;
   1:  PR[91,2] = PR[90,2] + 12.210;
   1:  PR[91,3] = PR[90,3] + 23.283;
   1:L PR[91] R[100]mm/sec CNT100;
   1:  PR[91,1] = PR[90,1] + -2.180;
   1:  PR[91,2] = PR[90,2] + 12.512;
   1:  PR[91,3] = PR[90,3] + 23.287;
   1:L PR[91] R[100]mm/sec CNT100;
   1:  PR[91,1] = PR[90,1] + -2.915;
   1:  PR[91,2] = PR[90,2] + 13.213;
   1:  PR[91,3] = PR[90,3] + 23.290;
   1:L PR[91] R[100]mm/sec CNT100;
   1:  PR[91,1] = PR[90,1] + -3.654;
   1:  PR[91,2] = PR[90,2] + 13.838;
   1:  PR[91,3] = PR[90,3] + 23.298;
   1:L PR[91] R[100]mm/sec CNT100;
   1:  PR[91,1] = PR[90,1] + -4.430;
   1:  PR[91,2] = PR[90,2] + 14.426;
   1:  PR[91,3] = PR[90,3] + 23.305;
   1:L PR[91] R[100]mm/sec CNT100;
   1:  PR[91,1] = PR[90,1] + -4.656;
   1:  PR[91,2] = PR[90,2] + 14.582;
   1:  PR[91,3] = PR[90,3] + 23.312;
   1:L PR[91] R[100]mm/sec CNT100;
   1:  PR[91,1] = PR[90,1] + -5.234;
   1:  PR[91,2] = PR[90,2] + 14.972;
   1:  PR[91,3] = PR[90,3] + 23.314;
   1:L PR[91] R[100]mm/sec CNT100;
   1:  PR[91,1] = PR[90,1] + -6.071;
   1:  PR[91,2] = PR[90,2] + 15.479;
   1:  PR[91,3] = PR[90,3] + 23.319;
   1:L PR[91] R[100]mm/sec CNT100;
   1:  PR[91,1] = PR[90,1] + -6.935;
   1:  PR[91,2] = PR[90,2] + 15.943;
   1:  PR[91,3] = PR[90,3] + 23.326;
   1:L PR[91] R[100]mm/sec CNT100;
   1:  PR[91,1] = PR[90,1] + -7.823;
   1:  PR[91,2] = PR[90,2] + 16.364;
   1:  PR[91,3] = PR[90,3] + 23.333;
   1:L PR[91] R[100]mm/sec CNT100;
   1:  PR[91,1] = PR[90,1] + -8.734;
   1:  PR[91,2] = PR[90,2] + 16.741;
   1:  PR[91,3] = PR[90,3] + 23.340;
   1:L PR[91] R[100]mm/sec CNT100;
   1:  PR[91,1] = PR[90,1] + -9.629;
   1:  PR[91,2] = PR[90,2] + 17.061;
   1:  PR[91,3] = PR[90,3] + 23.347;
   1:L PR[91] R[100]mm/sec CNT100;
   1:  PR[91,1] = PR[90,1] + -10.613;
   1:  PR[91,2] = PR[90,2] + 17.358;
   1:  PR[91,3] = PR[90,3] + 23.354;
   1:L PR[91] R[100]mm/sec CNT100;
   1:  PR[91,1] = PR[90,1] + -11.484;
   1:  PR[91,2] = PR[90,2] + 17.575;
   1:  PR[91,3] = PR[90,3] + 23.361;
   1:L PR[91] R[100]mm/sec CNT100;
   1:  PR[91,1] = PR[90,1] + -12.542;
   1:  PR[91,2] = PR[90,2] + 17.782;
   1:  PR[91,3] = PR[90,3] + 23.368;
   1:L PR[91] R[100]mm/sec CNT100;
   1:  PR[91,1] = PR[90,1] + -13.674;
   1:  PR[91,2] = PR[90,2] + 17.937;
   1:  PR[91,3] = PR[90,3] + 23.376;
   1:L PR[91] R[100]mm/sec CNT100;
   1:  PR[91,1] = PR[90,1] + -14.503;
   1:  PR[91,2] = PR[90,2] + 18.012;
   1:  PR[91,3] = PR[90,3] + 23.384;
   1:L PR[91] R[100]mm/sec CNT100;
   1:  PR[91,1] = PR[90,1] + -15.706;
   1:  PR[91,2] = PR[90,2] + 18.056;
   1:  PR[91,3] = PR[90,3] + 23.390;
   1:L PR[91] R[100]mm/sec CNT100;
   1:  PR[91,1] = PR[90,1] + -16.479;
   1:  PR[91,2] = PR[90,2] + 18.048;
   1:  PR[91,3] = PR[90,3] + 23.399;
   1:L PR[91] R[100]mm/sec CNT100;
   1:  PR[91,1] = PR[90,1] + -17.208;
   1:  PR[91,2] = PR[90,2] + 18.011;
   1:  PR[91,3] = PR[90,3] + 23.404;
   1:L PR[91] R[100]mm/sec CNT100;
   1:  PR[91,1] = PR[90,1] + -17.895;
   1:  PR[91,2] = PR[90,2] + 17.952;
   1:  PR[91,3] = PR[90,3] + 23.409;
   1:L PR[91] R[100]mm/sec CNT100;
   1:  PR[91,1] = PR[90,1] + -18.439;
   1:  PR[91,2] = PR[90,2] + 17.890;
   1:  PR[91,3] = PR[90,3] + 23.414;
   1:L PR[91] R[100]mm/sec CNT100;
   1:  PR[91,1] = PR[90,1] + -19.102;
   1:  PR[91,2] = PR[90,2] + 17.793;
   1:  PR[91,3] = PR[90,3] + 23.418;
   1:L PR[91] R[100]mm/sec CNT100;
   1:  PR[91,1] = PR[90,1] + -19.731;
   1:  PR[91,2] = PR[90,2] + 17.680;
   1:  PR[91,3] = PR[90,3] + 23.423;
   1:L PR[91] R[100]mm/sec CNT100;
   1:  PR[91,1] = PR[90,1] + -20.959;
   1:  PR[91,2] = PR[90,2] + 17.400;
   1:  PR[91,3] = PR[90,3] + 23.428;
   1:L PR[91] R[100]mm/sec CNT100;
   1:  PR[91,1] = PR[90,1] + -21.992;
   1:  PR[91,2] = PR[90,2] + 17.098;
   1:  PR[91,3] = PR[90,3] + 23.437;
   1:L PR[91] R[100]mm/sec CNT100;
   1:  PR[91,1] = PR[90,1] + -22.699;
   1:  PR[91,2] = PR[90,2] + 16.857;
   1:  PR[91,3] = PR[90,3] + 23.445;
   1:L PR[91] R[100]mm/sec CNT100;
   1:  PR[91,1] = PR[90,1] + -23.470;
   1:  PR[91,2] = PR[90,2] + 16.558;
   1:  PR[91,3] = PR[90,3] + 23.450;
   1:L PR[91] R[100]mm/sec CNT100;
   1:  PR[91,1] = PR[90,1] + -24.315;
   1:  PR[91,2] = PR[90,2] + 16.186;
   1:  PR[91,3] = PR[90,3] + 23.456;
   1:L PR[91] R[100]mm/sec CNT100;
   1:  PR[91,1] = PR[90,1] + -25.125;
   1:  PR[91,2] = PR[90,2] + 15.781;
   1:  PR[91,3] = PR[90,3] + 23.463;
   1:L PR[91] R[100]mm/sec CNT100;
   1:  PR[91,1] = PR[90,1] + -25.918;
   1:  PR[91,2] = PR[90,2] + 15.338;
   1:  PR[91,3] = PR[90,3] + 23.469;
   1:L PR[91] R[100]mm/sec CNT100;
   1:  PR[91,1] = PR[90,1] + -26.684;
   1:  PR[91,2] = PR[90,2] + 14.860;
   1:  PR[91,3] = PR[90,3] + 23.476;
   1:L PR[91] R[100]mm/sec CNT100;
   1:  PR[91,1] = PR[90,1] + -27.422;
   1:  PR[91,2] = PR[90,2] + 14.350;
   1:  PR[91,3] = PR[90,3] + 23.482;
   1:L PR[91] R[100]mm/sec CNT100;
   1:  PR[91,1] = PR[90,1] + -28.130;
   1:  PR[91,2] = PR[90,2] + 13.808;
   1:  PR[91,3] = PR[90,3] + 23.489;
   1:L PR[91] R[100]mm/sec CNT100;
   1:  PR[91,1] = PR[90,1] + -28.807;
   1:  PR[91,2] = PR[90,2] + 13.237;
   1:  PR[91,3] = PR[90,3] + 23.495;
   1:L PR[91] R[100]mm/sec CNT100;
   1:  PR[91,1] = PR[90,1] + -29.452;
   1:  PR[91,2] = PR[90,2] + 12.636;
   1:  PR[91,3] = PR[90,3] + 23.502;
   1:L PR[91] R[100]mm/sec CNT100;
   1:  PR[91,1] = PR[90,1] + -30.056;
   1:  PR[91,2] = PR[90,2] + 12.014;
   1:  PR[91,3] = PR[90,3] + 23.508;
   1:L PR[91] R[100]mm/sec CNT100;
   1:  PR[91,1] = PR[90,1] + -30.617;
   1:  PR[91,2] = PR[90,2] + 11.376;
   1:  PR[91,3] = PR[90,3] + 23.514;
   1:L PR[91] R[100]mm/sec CNT100;
   1:  PR[91,1] = PR[90,1] + -31.147;
   1:  PR[91,2] = PR[90,2] + 10.709;
   1:  PR[91,3] = PR[90,3] + 23.520;
   1:L PR[91] R[100]mm/sec CNT100;
   1:  PR[91,1] = PR[90,1] + -31.644;
   1:  PR[91,2] = PR[90,2] + 10.015;
   1:  PR[91,3] = PR[90,3] + 23.527;
   1:L PR[91] R[100]mm/sec CNT100;
   1:  PR[91,1] = PR[90,1] + -32.108;
   1:  PR[91,2] = PR[90,2] + 9.295;
   1:  PR[91,3] = PR[90,3] + 23.533;
   1:L PR[91] R[100]mm/sec CNT100;
   1:  PR[91,1] = PR[90,1] + -32.538;
   1:  PR[91,2] = PR[90,2] + 8.553;
   1:  PR[91,3] = PR[90,3] + 23.539;
   1:L PR[91] R[100]mm/sec CNT100;
   1:  PR[91,1] = PR[90,1] + -32.726;
   1:  PR[91,2] = PR[90,2] + 8.191;
   1:  PR[91,3] = PR[90,3] + 23.545;
   1:L PR[91] R[100]mm/sec CNT100;
   1:  PR[91,1] = PR[90,1] + -32.930;
   1:  PR[91,2] = PR[90,2] + 7.795;
   1:  PR[91,3] = PR[90,3] + 23.548;
   1:L PR[91] R[100]mm/sec CNT100;
   1:  PR[91,1] = PR[90,1] + -33.285;
   1:  PR[91,2] = PR[90,2] + 7.021;
   1:  PR[91,3] = PR[90,3] + 23.551;
   1:L PR[91] R[100]mm/sec CNT100;
   1:  PR[91,1] = PR[90,1] + -33.601;
   1:  PR[91,2] = PR[90,2] + 6.241;
   1:  PR[91,3] = PR[90,3] + 23.557;
   1:L PR[91] R[100]mm/sec CNT100;
   1:  PR[91,1] = PR[90,1] + -33.876;
   1:  PR[91,2] = PR[90,2] + 5.454;
   1:  PR[91,3] = PR[90,3] + 23.563;
   1:L PR[91] R[100]mm/sec CNT100;
   1:  PR[91,1] = PR[90,1] + -34.110;
   1:  PR[91,2] = PR[90,2] + 4.660;
   1:  PR[91,3] = PR[90,3] + 23.569;
   1:L PR[91] R[100]mm/sec CNT100;
   1:  PR[91,1] = PR[90,1] + -34.302;
   1:  PR[91,2] = PR[90,2] + 3.857;
   1:  PR[91,3] = PR[90,3] + 23.575;
   1:L PR[91] R[100]mm/sec CNT100;
   1:  PR[91,1] = PR[90,1] + -34.453;
   1:  PR[91,2] = PR[90,2] + 3.039;
   1:  PR[91,3] = PR[90,3] + 23.581;
   1:L PR[91] R[100]mm/sec CNT100;
   1:  PR[91,1] = PR[90,1] + -34.560;
   1:  PR[91,2] = PR[90,2] + 2.199;
   1:  PR[91,3] = PR[90,3] + 23.587;
   1:L PR[91] R[100]mm/sec CNT100;
   1:  PR[91,1] = PR[90,1] + -34.625;
   1:  PR[91,2] = PR[90,2] + 1.330;
   1:  PR[91,3] = PR[90,3] + 23.594;
   1:L PR[91] R[100]mm/sec CNT100;
   1:  PR[91,1] = PR[90,1] + -34.648;
   1:  PR[91,2] = PR[90,2] + 0.428;
   1:  PR[91,3] = PR[90,3] + 23.600;
   1:L PR[91] R[100]mm/sec CNT100;
   1:  PR[91,1] = PR[90,1] + -34.625;
   1:  PR[91,2] = PR[90,2] + -0.475;
   1:  PR[91,3] = PR[90,3] + 23.606;
   1:L PR[91] R[100]mm/sec CNT100;
   1:  PR[91,1] = PR[90,1] + -34.560;
   1:  PR[91,2] = PR[90,2] + -1.344;
   1:  PR[91,3] = PR[90,3] + 23.613;
   1:L PR[91] R[100]mm/sec CNT100;
   1:  PR[91,1] = PR[90,1] + -34.453;
   1:  PR[91,2] = PR[90,2] + -2.184;
   1:  PR[91,3] = PR[90,3] + 23.619;
   1:L PR[91] R[100]mm/sec CNT100;
   1:  PR[91,1] = PR[90,1] + -34.302;
   1:  PR[91,2] = PR[90,2] + -3.002;
   1:  PR[91,3] = PR[90,3] + 23.625;
   1:L PR[91] R[100]mm/sec CNT100;
   1:  PR[91,1] = PR[90,1] + -34.110;
   1:  PR[91,2] = PR[90,2] + -3.805;
   1:  PR[91,3] = PR[90,3] + 23.631;
   1:L PR[91] R[100]mm/sec CNT100;
   1:  PR[91,1] = PR[90,1] + -33.876;
   1:  PR[91,2] = PR[90,2] + -4.598;
   1:  PR[91,3] = PR[90,3] + 23.637;
   1:L PR[91] R[100]mm/sec CNT100;
   1:  PR[91,1] = PR[90,1] + -33.601;
   1:  PR[91,2] = PR[90,2] + -5.386;
   1:  PR[91,3] = PR[90,3] + 23.643;
   1:L PR[91] R[100]mm/sec CNT100;
   1:  PR[91,1] = PR[90,1] + -33.285;
   1:  PR[91,2] = PR[90,2] + -6.166;
   1:  PR[91,3] = PR[90,3] + 23.649;
   1:L PR[91] R[100]mm/sec CNT100;
   1:  PR[91,1] = PR[90,1] + -32.930;
   1:  PR[91,2] = PR[90,2] + -6.940;
   1:  PR[91,3] = PR[90,3] + 23.655;
   1:L PR[91] R[100]mm/sec CNT100;
   1:  PR[91,1] = PR[90,1] + -32.726;
   1:  PR[91,2] = PR[90,2] + -7.337;
   1:  PR[91,3] = PR[90,3] + 23.661;
   1:L PR[91] R[100]mm/sec CNT100;
   1:  PR[91,1] = PR[90,1] + -32.538;
   1:  PR[91,2] = PR[90,2] + -7.697;
   1:  PR[91,3] = PR[90,3] + 23.665;
   1:L PR[91] R[100]mm/sec CNT100;
   1:  PR[91,1] = PR[90,1] + -32.108;
   1:  PR[91,2] = PR[90,2] + -8.440;
   1:  PR[91,3] = PR[90,3] + 23.668;
   1:L PR[91] R[100]mm/sec CNT100;
   1:  PR[91,1] = PR[90,1] + -31.644;
   1:  PR[91,2] = PR[90,2] + -9.159;
   1:  PR[91,3] = PR[90,3] + 23.674;
   1:L PR[91] R[100]mm/sec CNT100;
   1:  PR[91,1] = PR[90,1] + -31.147;
   1:  PR[91,2] = PR[90,2] + -9.854;
   1:  PR[91,3] = PR[90,3] + 23.680;
   1:L PR[91] R[100]mm/sec CNT100;
   1:  PR[91,1] = PR[90,1] + -30.617;
   1:  PR[91,2] = PR[90,2] + -10.521;
   1:  PR[91,3] = PR[90,3] + 23.686;
   1:L PR[91] R[100]mm/sec CNT100;
   1:  PR[91,1] = PR[90,1] + -30.056;
   1:  PR[91,2] = PR[90,2] + -11.159;
   1:  PR[91,3] = PR[90,3] + 23.692;
   1:L PR[91] R[100]mm/sec CNT100;
   1:  PR[91,1] = PR[90,1] + -29.452;
   1:  PR[91,2] = PR[90,2] + -11.781;
   1:  PR[91,3] = PR[90,3] + 23.698;
   1:L PR[91] R[100]mm/sec CNT100;
   1:  PR[91,1] = PR[90,1] + -28.807;
   1:  PR[91,2] = PR[90,2] + -12.381;
   1:  PR[91,3] = PR[90,3] + 23.705;
   1:L PR[91] R[100]mm/sec CNT100;
   1:  PR[91,1] = PR[90,1] + -28.130;
   1:  PR[91,2] = PR[90,2] + -12.953;
   1:  PR[91,3] = PR[90,3] + 23.711;
   1:L PR[91] R[100]mm/sec CNT100;
   1:  PR[91,1] = PR[90,1] + -27.421;
   1:  PR[91,2] = PR[90,2] + -13.495;
   1:  PR[91,3] = PR[90,3] + 23.717;
   1:L PR[91] R[100]mm/sec CNT100;
   1:  PR[91,1] = PR[90,1] + -27.055;
   1:  PR[91,2] = PR[90,2] + -13.750;
   1:  PR[91,3] = PR[90,3] + 23.724;
   1:L PR[91] R[100]mm/sec CNT100;
   1:  PR[91,1] = PR[90,1] + -26.684;
   1:  PR[91,2] = PR[90,2] + -14.004;
   1:  PR[91,3] = PR[90,3] + 23.727;
   1:L PR[91] R[100]mm/sec CNT100;
   1:  PR[91,1] = PR[90,1] + -25.918;
   1:  PR[91,2] = PR[90,2] + -14.482;
   1:  PR[91,3] = PR[90,3] + 23.730;
   1:L PR[91] R[100]mm/sec CNT100;
   1:  PR[91,1] = PR[90,1] + -25.126;
   1:  PR[91,2] = PR[90,2] + -14.926;
   1:  PR[91,3] = PR[90,3] + 23.737;
   1:L PR[91] R[100]mm/sec CNT100;
   1:  PR[91,1] = PR[90,1] + -24.303;
   1:  PR[91,2] = PR[90,2] + -15.336;
   1:  PR[91,3] = PR[90,3] + 23.743;
   1:L PR[91] R[100]mm/sec CNT100;
   1:  PR[91,1] = PR[90,1] + -23.470;
   1:  PR[91,2] = PR[90,2] + -15.703;
   1:  PR[91,3] = PR[90,3] + 23.750;
   1:L PR[91] R[100]mm/sec CNT100;
   1:  PR[91,1] = PR[90,1] + -22.701;
   1:  PR[91,2] = PR[90,2] + -16.001;
   1:  PR[91,3] = PR[90,3] + 23.757;
   1:L PR[91] R[100]mm/sec CNT100;
   1:  PR[91,1] = PR[90,1] + -21.676;
   1:  PR[91,2] = PR[90,2] + -16.342;
   1:  PR[91,3] = PR[90,3] + 23.763;
   1:L PR[91] R[100]mm/sec CNT100;
   1:  PR[91,1] = PR[90,1] + -20.957;
   1:  PR[91,2] = PR[90,2] + -16.545;
   1:  PR[91,3] = PR[90,3] + 23.770;
   1:L PR[91] R[100]mm/sec CNT100;
   1:  PR[91,1] = PR[90,1] + -20.308;
   1:  PR[91,2] = PR[90,2] + -16.703;
   1:  PR[91,3] = PR[90,3] + 23.776;
   1:L PR[91] R[100]mm/sec CNT100;
   1:  PR[91,1] = PR[90,1] + -19.098;
   1:  PR[91,2] = PR[90,2] + -16.938;
   1:  PR[91,3] = PR[90,3] + 23.781;
   1:L PR[91] R[100]mm/sec CNT100;
   1:  PR[91,1] = PR[90,1] + -18.440;
   1:  PR[91,2] = PR[90,2] + -17.035;
   1:  PR[91,3] = PR[90,3] + 23.790;
   1:L PR[91] R[100]mm/sec CNT100;
   1:  PR[91,1] = PR[90,1] + -17.736;
   1:  PR[91,2] = PR[90,2] + -17.113;
   1:  PR[91,3] = PR[90,3] + 23.794;
   1:L PR[91] R[100]mm/sec CNT100;
   1:  PR[91,1] = PR[90,1] + -16.478;
   1:  PR[91,2] = PR[90,2] + -17.192;
   1:  PR[91,3] = PR[90,3] + 23.799;
   1:L PR[91] R[100]mm/sec CNT100;
   1:  PR[91,1] = PR[90,1] + -15.292;
   1:  PR[91,2] = PR[90,2] + -17.194;
   1:  PR[91,3] = PR[90,3] + 23.809;
   1:L PR[91] R[100]mm/sec CNT100;
   1:  PR[91,1] = PR[90,1] + -14.507;
   1:  PR[91,2] = PR[90,2] + -17.157;
   1:  PR[91,3] = PR[90,3] + 23.817;
   1:L PR[91] R[100]mm/sec CNT100;
   1:  PR[91,1] = PR[90,1] + -13.675;
   1:  PR[91,2] = PR[90,2] + -17.082;
   1:  PR[91,3] = PR[90,3] + 23.823;
   1:L PR[91] R[100]mm/sec CNT100;
   1:  PR[91,1] = PR[90,1] + -12.543;
   1:  PR[91,2] = PR[90,2] + -16.927;
   1:  PR[91,3] = PR[90,3] + 23.829;
   1:L PR[91] R[100]mm/sec CNT100;
   1:  PR[91,1] = PR[90,1] + -11.486;
   1:  PR[91,2] = PR[90,2] + -16.720;
   1:  PR[91,3] = PR[90,3] + 23.837;
   1:L PR[91] R[100]mm/sec CNT100;
   1:  PR[91,1] = PR[90,1] + -10.494;
   1:  PR[91,2] = PR[90,2] + -16.469;
   1:  PR[91,3] = PR[90,3] + 23.845;
   1:L PR[91] R[100]mm/sec CNT100;
   1:  PR[91,1] = PR[90,1] + -9.630;
   1:  PR[91,2] = PR[90,2] + -16.207;
   1:  PR[91,3] = PR[90,3] + 23.852;
   1:L PR[91] R[100]mm/sec CNT100;
   1:  PR[91,1] = PR[90,1] + -8.712;
   1:  PR[91,2] = PR[90,2] + -15.877;
   1:  PR[91,3] = PR[90,3] + 23.859;
   1:L PR[91] R[100]mm/sec CNT100;
   1:  PR[91,1] = PR[90,1] + -7.824;
   1:  PR[91,2] = PR[90,2] + -15.509;
   1:  PR[91,3] = PR[90,3] + 23.866;
   1:L PR[91] R[100]mm/sec CNT100;
   1:  PR[91,1] = PR[90,1] + -6.936;
   1:  PR[91,2] = PR[90,2] + -15.089;
   1:  PR[91,3] = PR[90,3] + 23.873;
   1:L PR[91] R[100]mm/sec CNT100;
   1:  PR[91,1] = PR[90,1] + -6.072;
   1:  PR[91,2] = PR[90,2] + -14.624;
   1:  PR[91,3] = PR[90,3] + 23.880;
   1:L PR[91] R[100]mm/sec CNT100;
   1:  PR[91,1] = PR[90,1] + -5.235;
   1:  PR[91,2] = PR[90,2] + -14.118;
   1:  PR[91,3] = PR[90,3] + 23.887;
   1:L PR[91] R[100]mm/sec CNT100;
   1:  PR[91,1] = PR[90,1] + -4.657;
   1:  PR[91,2] = PR[90,2] + -13.727;
   1:  PR[91,3] = PR[90,3] + 23.894;
   1:L PR[91] R[100]mm/sec CNT100;
   1:  PR[91,1] = PR[90,1] + -4.430;
   1:  PR[91,2] = PR[90,2] + -13.572;
   1:  PR[91,3] = PR[90,3] + 23.899;
   1:L PR[91] R[100]mm/sec CNT100;
   1:  PR[91,1] = PR[90,1] + -3.655;
   1:  PR[91,2] = PR[90,2] + -12.983;
   1:  PR[91,3] = PR[90,3] + 23.901;
   1:L PR[91] R[100]mm/sec CNT100;
   1:  PR[91,1] = PR[90,1] + -2.916;
   1:  PR[91,2] = PR[90,2] + -12.358;
   1:  PR[91,3] = PR[90,3] + 23.908;
   1:L PR[91] R[100]mm/sec CNT100;
   1:  PR[91,1] = PR[90,1] + -2.179;
   1:  PR[91,2] = PR[90,2] + -11.656;
   1:  PR[91,3] = PR[90,3] + 23.915;
   1:L PR[91] R[100]mm/sec CNT100;
   1:  PR[91,1] = PR[90,1] + -1.824;
   1:  PR[91,2] = PR[90,2] + -11.355;
   1:  PR[91,3] = PR[90,3] + 23.922;
   1:L PR[91] R[100]mm/sec CNT100;
   1:  PR[91,1] = PR[90,1] + -1.402;
   1:  PR[91,2] = PR[90,2] + -11.097;
   1:  PR[91,3] = PR[90,3] + 23.926;
   1:L PR[91] R[100]mm/sec CNT100;
   1:  PR[91,1] = PR[90,1] + -0.940;
   1:  PR[91,2] = PR[90,2] + -10.911;
   1:  PR[91,3] = PR[90,3] + 23.929;
   1:L PR[91] R[100]mm/sec CNT100;
   1:  PR[91,1] = PR[90,1] + -0.456;
   1:  PR[91,2] = PR[90,2] + -10.812;
   1:  PR[91,3] = PR[90,3] + 23.933;
   1:L PR[91] R[100]mm/sec CNT100;
   1:  PR[91,1] = PR[90,1] + 0.042;
   1:  PR[91,2] = PR[90,2] + -10.793;
   1:  PR[91,3] = PR[90,3] + 23.936;
   1:L PR[91] R[100]mm/sec CNT100;
   1:  PR[91] = PR[90];
   1:  PR[91,1] = PR[90,1] + 0.646;
   1:  PR[91,2] = PR[90,2] + -11.564;
   1:  PR[91,3] = PR[90,3] + 25.270;
   1:L PR[91] R[100]mm/sec CNT100;
   1:  PR[91,1] = PR[90,1] + 1.116;
   1:  PR[91,2] = PR[90,2] + -11.743;
   1:  PR[91,3] = PR[90,3] + 23.944;
   1:L PR[91] R[100]mm/sec CNT100;
   1:  PR[91,1] = PR[90,1] + 1.557;
   1:  PR[91,2] = PR[90,2] + -11.996;
   1:  PR[91,3] = PR[90,3] + 23.947;
   1:L PR[91] R[100]mm/sec CNT100;
   1:  PR[91,1] = PR[90,1] + 2.773;
   1:  PR[91,2] = PR[90,2] + -13.037;
   1:  PR[91,3] = PR[90,3] + 23.951;
   1:L PR[91] R[100]mm/sec CNT100;
   1:  PR[91,1] = PR[90,1] + 3.539;
   1:  PR[91,2] = PR[90,2] + -13.624;
   1:  PR[91,3] = PR[90,3] + 23.963;
   1:L PR[91] R[100]mm/sec CNT100;
   1:  PR[91,1] = PR[90,1] + 4.337;
   1:  PR[91,2] = PR[90,2] + -14.172;
   1:  PR[91,3] = PR[90,3] + 23.970;
   1:L PR[91] R[100]mm/sec CNT100;
   1:  PR[91,1] = PR[90,1] + 5.168;
   1:  PR[91,2] = PR[90,2] + -14.681;
   1:  PR[91,3] = PR[90,3] + 23.977;
   1:L PR[91] R[100]mm/sec CNT100;
   1:  PR[91,1] = PR[90,1] + 6.028;
   1:  PR[91,2] = PR[90,2] + -15.149;
   1:  PR[91,3] = PR[90,3] + 23.984;
   1:L PR[91] R[100]mm/sec CNT100;
   1:  PR[91,1] = PR[90,1] + 6.916;
   1:  PR[91,2] = PR[90,2] + -15.575;
   1:  PR[91,3] = PR[90,3] + 23.991;
   1:L PR[91] R[100]mm/sec CNT100;
   1:  PR[91,1] = PR[90,1] + 7.830;
   1:  PR[91,2] = PR[90,2] + -15.957;
   1:  PR[91,3] = PR[90,3] + 23.998;
   1:L PR[91] R[100]mm/sec CNT100;
   1:  PR[91,1] = PR[90,1] + 8.767;
   1:  PR[91,2] = PR[90,2] + -16.295;
   1:  PR[91,3] = PR[90,3] + 24.006;
   1:L PR[91] R[100]mm/sec CNT100;
   1:  PR[91,1] = PR[90,1] + 9.725;
   1:  PR[91,2] = PR[90,2] + -16.586;
   1:  PR[91,3] = PR[90,3] + 24.013;
   1:L PR[91] R[100]mm/sec CNT100;
   1:  PR[91,1] = PR[90,1] + 10.700;
   1:  PR[91,2] = PR[90,2] + -16.829;
   1:  PR[91,3] = PR[90,3] + 24.020;
   1:L PR[91] R[100]mm/sec CNT100;
   1:  PR[91,1] = PR[90,1] + 11.691;
   1:  PR[91,2] = PR[90,2] + -17.024;
   1:  PR[91,3] = PR[90,3] + 24.028;
   1:L PR[91] R[100]mm/sec CNT100;
   1:  PR[91,1] = PR[90,1] + 12.727;
   1:  PR[91,2] = PR[90,2] + -17.172;
   1:  PR[91,3] = PR[90,3] + 24.035;
   1:L PR[91] R[100]mm/sec CNT100;
   1:  PR[91,1] = PR[90,1] + 13.695;
   1:  PR[91,2] = PR[90,2] + -17.262;
   1:  PR[91,3] = PR[90,3] + 24.043;
   1:L PR[91] R[100]mm/sec CNT100;
   1:  PR[91,1] = PR[90,1] + 14.642;
   1:  PR[91,2] = PR[90,2] + -17.305;
   1:  PR[91,3] = PR[90,3] + 24.050;
   1:L PR[91] R[100]mm/sec CNT100;
   1:  PR[91,1] = PR[90,1] + 15.676;
   1:  PR[91,2] = PR[90,2] + -17.301;
   1:  PR[91,3] = PR[90,3] + 24.057;
   1:L PR[91] R[100]mm/sec CNT100;
   1:  PR[91,1] = PR[90,1] + 16.768;
   1:  PR[91,2] = PR[90,2] + -17.239;
   1:  PR[91,3] = PR[90,3] + 24.064;
   1:L PR[91] R[100]mm/sec CNT100;
   1:  PR[91,1] = PR[90,1] + 17.644;
   1:  PR[91,2] = PR[90,2] + -17.147;
   1:  PR[91,3] = PR[90,3] + 24.072;
   1:L PR[91] R[100]mm/sec CNT100;
   1:  PR[91,1] = PR[90,1] + 18.462;
   1:  PR[91,2] = PR[90,2] + -17.025;
   1:  PR[91,3] = PR[90,3] + 24.079;
   1:L PR[91] R[100]mm/sec CNT100;
   1:  PR[91,1] = PR[90,1] + 19.579;
   1:  PR[91,2] = PR[90,2] + -16.803;
   1:  PR[91,3] = PR[90,3] + 24.085;
   1:L PR[91] R[100]mm/sec CNT100;
   1:  PR[91,1] = PR[90,1] + 20.320;
   1:  PR[91,2] = PR[90,2] + -16.617;
   1:  PR[91,3] = PR[90,3] + 24.093;
   1:L PR[91] R[100]mm/sec CNT100;
   1:  PR[91,1] = PR[90,1] + 21.460;
   1:  PR[91,2] = PR[90,2] + -16.273;
   1:  PR[91,3] = PR[90,3] + 24.099;
   1:L PR[91] R[100]mm/sec CNT100;
   1:  PR[91,1] = PR[90,1] + 22.124;
   1:  PR[91,2] = PR[90,2] + -16.038;
   1:  PR[91,3] = PR[90,3] + 24.107;
   1:L PR[91] R[100]mm/sec CNT100;
   1:  PR[91,1] = PR[90,1] + 23.275;
   1:  PR[91,2] = PR[90,2] + -15.566;
   1:  PR[91,3] = PR[90,3] + 24.112;
   1:L PR[91] R[100]mm/sec CNT100;
   1:  PR[91,1] = PR[90,1] + 23.863;
   1:  PR[91,2] = PR[90,2] + -15.292;
   1:  PR[91,3] = PR[90,3] + 24.121;
   1:L PR[91] R[100]mm/sec CNT100;
   1:  PR[91,1] = PR[90,1] + 24.425;
   1:  PR[91,2] = PR[90,2] + -15.008;
   1:  PR[91,3] = PR[90,3] + 24.126;
   1:L PR[91] R[100]mm/sec CNT100;
   1:  PR[91,1] = PR[90,1] + 25.449;
   1:  PR[91,2] = PR[90,2] + -14.428;
   1:  PR[91,3] = PR[90,3] + 24.131;
   1:L PR[91] R[100]mm/sec CNT100;
   1:  PR[91,1] = PR[90,1] + 26.031;
   1:  PR[91,2] = PR[90,2] + -14.061;
   1:  PR[91,3] = PR[90,3] + 24.139;
   1:L PR[91] R[100]mm/sec CNT100;
   1:  PR[91,1] = PR[90,1] + 26.648;
   1:  PR[91,2] = PR[90,2] + -13.638;
   1:  PR[91,3] = PR[90,3] + 24.144;
   1:L PR[91] R[100]mm/sec CNT100;
   1:  PR[91,1] = PR[90,1] + 27.472;
   1:  PR[91,2] = PR[90,2] + -13.013;
   1:  PR[91,3] = PR[90,3] + 24.150;
   1:L PR[91] R[100]mm/sec CNT100;
   1:  PR[91,1] = PR[90,1] + 28.087;
   1:  PR[91,2] = PR[90,2] + -12.497;
   1:  PR[91,3] = PR[90,3] + 24.157;
   1:L PR[91] R[100]mm/sec CNT100;
   1:  PR[91,1] = PR[90,1] + 28.764;
   1:  PR[91,2] = PR[90,2] + -11.871;
   1:  PR[91,3] = PR[90,3] + 24.163;
   1:L PR[91] R[100]mm/sec CNT100;
   1:  PR[91,1] = PR[90,1] + 29.364;
   1:  PR[91,2] = PR[90,2] + -11.258;
   1:  PR[91,3] = PR[90,3] + 24.170;
   1:L PR[91] R[100]mm/sec CNT100;
   1:  PR[91,1] = PR[90,1] + 29.949;
   1:  PR[91,2] = PR[90,2] + -10.594;
   1:  PR[91,3] = PR[90,3] + 24.176;
   1:L PR[91] R[100]mm/sec CNT100;
   1:  PR[91,1] = PR[90,1] + 30.499;
   1:  PR[91,2] = PR[90,2] + -9.904;
   1:  PR[91,3] = PR[90,3] + 24.183;
   1:L PR[91] R[100]mm/sec CNT100;
   1:  PR[91,1] = PR[90,1] + 31.012;
   1:  PR[91,2] = PR[90,2] + -9.190;
   1:  PR[91,3] = PR[90,3] + 24.189;
   1:L PR[91] R[100]mm/sec CNT100;
   1:  PR[91,1] = PR[90,1] + 31.488;
   1:  PR[91,2] = PR[90,2] + -8.455;
   1:  PR[91,3] = PR[90,3] + 24.196;
   1:L PR[91] R[100]mm/sec CNT100;
   1:  PR[91,1] = PR[90,1] + 31.926;
   1:  PR[91,2] = PR[90,2] + -7.703;
   1:  PR[91,3] = PR[90,3] + 24.202;
   1:L PR[91] R[100]mm/sec CNT100;
   1:  PR[91,1] = PR[90,1] + 32.325;
   1:  PR[91,2] = PR[90,2] + -6.938;
   1:  PR[91,3] = PR[90,3] + 24.208;
   1:L PR[91] R[100]mm/sec CNT100;
   1:  PR[91,1] = PR[90,1] + 32.683;
   1:  PR[91,2] = PR[90,2] + -6.165;
   1:  PR[91,3] = PR[90,3] + 24.215;
   1:L PR[91] R[100]mm/sec CNT100;
   1:  PR[91,1] = PR[90,1] + 33.000;
   1:  PR[91,2] = PR[90,2] + -5.387;
   1:  PR[91,3] = PR[90,3] + 24.221;
   1:L PR[91] R[100]mm/sec CNT100;
   1:  PR[91,1] = PR[90,1] + 33.275;
   1:  PR[91,2] = PR[90,2] + -4.603;
   1:  PR[91,3] = PR[90,3] + 24.227;
   1:L PR[91] R[100]mm/sec CNT100;
   1:  PR[91,1] = PR[90,1] + 33.508;
   1:  PR[91,2] = PR[90,2] + -3.811;
   1:  PR[91,3] = PR[90,3] + 24.233;
   1:L PR[91] R[100]mm/sec CNT100;
   1:  PR[91,1] = PR[90,1] + 33.700;
   1:  PR[91,2] = PR[90,2] + -3.008;
   1:  PR[91,3] = PR[90,3] + 24.239;
   1:L PR[91] R[100]mm/sec CNT100;
   1:  PR[91,1] = PR[90,1] + 33.849;
   1:  PR[91,2] = PR[90,2] + -2.188;
   1:  PR[91,3] = PR[90,3] + 24.245;
   1:L PR[91] R[100]mm/sec CNT100;
   1:  PR[91,1] = PR[90,1] + 33.956;
   1:  PR[91,2] = PR[90,2] + -1.345;
   1:  PR[91,3] = PR[90,3] + 24.251;
   1:L PR[91] R[100]mm/sec CNT100;
   1:  PR[91,1] = PR[90,1] + 34.021;
   1:  PR[91,2] = PR[90,2] + -0.475;
   1:  PR[91,3] = PR[90,3] + 24.258;
   1:L PR[91] R[100]mm/sec CNT100;
   1:  PR[91,1] = PR[90,1] + 34.044;
   1:  PR[91,2] = PR[90,2] + 0.428;
   1:  PR[91,3] = PR[90,3] + 24.264;
   1:L PR[91] R[100]mm/sec CNT100;
   1:  PR[91,1] = PR[90,1] + 34.021;
   1:  PR[91,2] = PR[90,2] + 1.330;
   1:  PR[91,3] = PR[90,3] + 24.271;
   1:L PR[91] R[100]mm/sec CNT100;
   1:  PR[91,1] = PR[90,1] + 33.956;
   1:  PR[91,2] = PR[90,2] + 2.200;
   1:  PR[91,3] = PR[90,3] + 24.277;
   1:L PR[91] R[100]mm/sec CNT100;
   1:  PR[91,1] = PR[90,1] + 33.849;
   1:  PR[91,2] = PR[90,2] + 3.043;
   1:  PR[91,3] = PR[90,3] + 24.283;
   1:L PR[91] R[100]mm/sec CNT100;
   1:  PR[91,1] = PR[90,1] + 33.700;
   1:  PR[91,2] = PR[90,2] + 3.863;
   1:  PR[91,3] = PR[90,3] + 24.290;
   1:L PR[91] R[100]mm/sec CNT100;
   1:  PR[91,1] = PR[90,1] + 33.508;
   1:  PR[91,2] = PR[90,2] + 4.666;
   1:  PR[91,3] = PR[90,3] + 24.296;
   1:L PR[91] R[100]mm/sec CNT100;
   1:  PR[91,1] = PR[90,1] + 33.275;
   1:  PR[91,2] = PR[90,2] + 5.458;
   1:  PR[91,3] = PR[90,3] + 24.302;
   1:L PR[91] R[100]mm/sec CNT100;
   1:  PR[91,1] = PR[90,1] + 33.000;
   1:  PR[91,2] = PR[90,2] + 6.242;
   1:  PR[91,3] = PR[90,3] + 24.308;
   1:L PR[91] R[100]mm/sec CNT100;
   1:  PR[91,1] = PR[90,1] + 32.683;
   1:  PR[91,2] = PR[90,2] + 7.020;
   1:  PR[91,3] = PR[90,3] + 24.314;
   1:L PR[91] R[100]mm/sec CNT100;
   1:  PR[91,1] = PR[90,1] + 32.325;
   1:  PR[91,2] = PR[90,2] + 7.793;
   1:  PR[91,3] = PR[90,3] + 24.320;
   1:L PR[91] R[100]mm/sec CNT100;
   1:  PR[91,1] = PR[90,1] + 31.926;
   1:  PR[91,2] = PR[90,2] + 8.558;
   1:  PR[91,3] = PR[90,3] + 24.326;
   1:L PR[91] R[100]mm/sec CNT100;
   1:  PR[91,1] = PR[90,1] + 31.488;
   1:  PR[91,2] = PR[90,2] + 9.310;
   1:  PR[91,3] = PR[90,3] + 24.333;
   1:L PR[91] R[100]mm/sec CNT100;
   1:  PR[91,1] = PR[90,1] + 31.012;
   1:  PR[91,2] = PR[90,2] + 10.045;
   1:  PR[91,3] = PR[90,3] + 24.339;
   1:L PR[91] R[100]mm/sec CNT100;
   1:  PR[91,1] = PR[90,1] + 30.499;
   1:  PR[91,2] = PR[90,2] + 10.759;
   1:  PR[91,3] = PR[90,3] + 24.345;
   1:L PR[91] R[100]mm/sec CNT100;
   1:  PR[91,1] = PR[90,1] + 29.949;
   1:  PR[91,2] = PR[90,2] + 11.450;
   1:  PR[91,3] = PR[90,3] + 24.352;
   1:L PR[91] R[100]mm/sec CNT100;
   1:  PR[91,1] = PR[90,1] + 29.364;
   1:  PR[91,2] = PR[90,2] + 12.113;
   1:  PR[91,3] = PR[90,3] + 24.358;
   1:L PR[91] R[100]mm/sec CNT100;
   1:  PR[91,1] = PR[90,1] + 28.764;
   1:  PR[91,2] = PR[90,2] + 12.727;
   1:  PR[91,3] = PR[90,3] + 24.365;
   1:L PR[91] R[100]mm/sec CNT100;
   1:  PR[91,1] = PR[90,1] + 28.088;
   1:  PR[91,2] = PR[90,2] + 13.351;
   1:  PR[91,3] = PR[90,3] + 24.371;
   1:L PR[91] R[100]mm/sec CNT100;
   1:  PR[91,1] = PR[90,1] + 27.298;
   1:  PR[91,2] = PR[90,2] + 14.005;
   1:  PR[91,3] = PR[90,3] + 24.378;
   1:L PR[91] R[100]mm/sec CNT100;
   1:  PR[91,1] = PR[90,1] + 26.649;
   1:  PR[91,2] = PR[90,2] + 14.492;
   1:  PR[91,3] = PR[90,3] + 24.385;
   1:L PR[91] R[100]mm/sec CNT100;
   1:  PR[91,1] = PR[90,1] + 26.034;
   1:  PR[91,2] = PR[90,2] + 14.914;
   1:  PR[91,3] = PR[90,3] + 24.391;
   1:L PR[91] R[100]mm/sec CNT100;
   1:  PR[91,1] = PR[90,1] + 25.029;
   1:  PR[91,2] = PR[90,2] + 15.531;
   1:  PR[91,3] = PR[90,3] + 24.397;
   1:L PR[91] R[100]mm/sec CNT100;
   1:  PR[91,1] = PR[90,1] + 24.429;
   1:  PR[91,2] = PR[90,2] + 15.861;
   1:  PR[91,3] = PR[90,3] + 24.405;
   1:L PR[91] R[100]mm/sec CNT100;
   1:  PR[91,1] = PR[90,1] + 23.863;
   1:  PR[91,2] = PR[90,2] + 16.147;
   1:  PR[91,3] = PR[90,3] + 24.410;
   1:L PR[91] R[100]mm/sec CNT100;
   1:  PR[91,1] = PR[90,1] + 23.272;
   1:  PR[91,2] = PR[90,2] + 16.423;
   1:  PR[91,3] = PR[90,3] + 24.415;
   1:L PR[91] R[100]mm/sec CNT100;
   1:  PR[91,1] = PR[90,1] + 22.637;
   1:  PR[91,2] = PR[90,2] + 16.693;
   1:  PR[91,3] = PR[90,3] + 24.420;
   1:L PR[91] R[100]mm/sec CNT100;
   1:  PR[91,1] = PR[90,1] + 21.456;
   1:  PR[91,2] = PR[90,2] + 17.130;
   1:  PR[91,3] = PR[90,3] + 24.425;
   1:L PR[91] R[100]mm/sec CNT100;
   1:  PR[91,1] = PR[90,1] + 20.320;
   1:  PR[91,2] = PR[90,2] + 17.472;
   1:  PR[91,3] = PR[90,3] + 24.434;
   1:L PR[91] R[100]mm/sec CNT100;
   1:  PR[91,1] = PR[90,1] + 19.578;
   1:  PR[91,2] = PR[90,2] + 17.658;
   1:  PR[91,3] = PR[90,3] + 24.443;
   1:L PR[91] R[100]mm/sec CNT100;
   1:  PR[91,1] = PR[90,1] + 18.462;
   1:  PR[91,2] = PR[90,2] + 17.880;
   1:  PR[91,3] = PR[90,3] + 24.448;
   1:L PR[91] R[100]mm/sec CNT100;
   1:  PR[91,1] = PR[90,1] + 17.644;
   1:  PR[91,2] = PR[90,2] + 18.003;
   1:  PR[91,3] = PR[90,3] + 24.456;
   1:L PR[91] R[100]mm/sec CNT100;
   1:  PR[91,1] = PR[90,1] + 16.768;
   1:  PR[91,2] = PR[90,2] + 18.094;
   1:  PR[91,3] = PR[90,3] + 24.462;
   1:L PR[91] R[100]mm/sec CNT100;
   1:  PR[91,1] = PR[90,1] + 15.675;
   1:  PR[91,2] = PR[90,2] + 18.156;
   1:  PR[91,3] = PR[90,3] + 24.469;
   1:L PR[91] R[100]mm/sec CNT100;
   1:  PR[91,1] = PR[90,1] + 14.641;
   1:  PR[91,2] = PR[90,2] + 18.160;
   1:  PR[91,3] = PR[90,3] + 24.477;
   1:L PR[91] R[100]mm/sec CNT100;
   1:  PR[91,1] = PR[90,1] + 13.694;
   1:  PR[91,2] = PR[90,2] + 18.117;
   1:  PR[91,3] = PR[90,3] + 24.484;
   1:L PR[91] R[100]mm/sec CNT100;
   1:  PR[91,1] = PR[90,1] + 12.695;
   1:  PR[91,2] = PR[90,2] + 18.023;
   1:  PR[91,3] = PR[90,3] + 24.491;
   1:L PR[91] R[100]mm/sec CNT100;
   1:  PR[91,1] = PR[90,1] + 11.691;
   1:  PR[91,2] = PR[90,2] + 17.879;
   1:  PR[91,3] = PR[90,3] + 24.499;
   1:L PR[91] R[100]mm/sec CNT100;
   1:  PR[91,1] = PR[90,1] + 10.700;
   1:  PR[91,2] = PR[90,2] + 17.684;
   1:  PR[91,3] = PR[90,3] + 24.506;
   1:L PR[91] R[100]mm/sec CNT100;
   1:  PR[91,1] = PR[90,1] + 9.725;
   1:  PR[91,2] = PR[90,2] + 17.441;
   1:  PR[91,3] = PR[90,3] + 24.513;
   1:L PR[91] R[100]mm/sec CNT100;
   1:  PR[91,1] = PR[90,1] + 8.765;
   1:  PR[91,2] = PR[90,2] + 17.149;
   1:  PR[91,3] = PR[90,3] + 24.521;
   1:L PR[91] R[100]mm/sec CNT100;
   1:  PR[91,1] = PR[90,1] + 8.199;
   1:  PR[91,2] = PR[90,2] + 16.949;
   1:  PR[91,3] = PR[90,3] + 24.528;
   1:L PR[91] R[100]mm/sec CNT100;
   1:  PR[91,1] = PR[90,1] + 7.833;
   1:  PR[91,2] = PR[90,2] + 16.813;
   1:  PR[91,3] = PR[90,3] + 24.533;
   1:L PR[91] R[100]mm/sec CNT100;
   1:  PR[91,1] = PR[90,1] + 6.916;
   1:  PR[91,2] = PR[90,2] + 16.430;
   1:  PR[91,3] = PR[90,3] + 24.535;
   1:L PR[91] R[100]mm/sec CNT100;
   1:  PR[91,1] = PR[90,1] + 6.028;
   1:  PR[91,2] = PR[90,2] + 16.004;
   1:  PR[91,3] = PR[90,3] + 24.543;
   1:L PR[91] R[100]mm/sec CNT100;
   1:  PR[91,1] = PR[90,1] + 5.165;
   1:  PR[91,2] = PR[90,2] + 15.535;
   1:  PR[91,3] = PR[90,3] + 24.550;
   1:L PR[91] R[100]mm/sec CNT100;
   1:  PR[91,1] = PR[90,1] + 4.885;
   1:  PR[91,2] = PR[90,2] + 15.366;
   1:  PR[91,3] = PR[90,3] + 24.557;
   1:L PR[91] R[100]mm/sec CNT100;
   1:  PR[91,1] = PR[90,1] + 4.338;
   1:  PR[91,2] = PR[90,2] + 15.028;
   1:  PR[91,3] = PR[90,3] + 24.559;
   1:L PR[91] R[100]mm/sec CNT100;
   1:  PR[91,1] = PR[90,1] + 3.539;
   1:  PR[91,2] = PR[90,2] + 14.479;
   1:  PR[91,3] = PR[90,3] + 24.564;
   1:L PR[91] R[100]mm/sec CNT100;
   1:  PR[91,1] = PR[90,1] + 2.774;
   1:  PR[91,2] = PR[90,2] + 13.893;
   1:  PR[91,3] = PR[90,3] + 24.571;
   1:L PR[91] R[100]mm/sec CNT100;
   1:  PR[91,1] = PR[90,1] + 1.557;
   1:  PR[91,2] = PR[90,2] + 12.851;
   1:  PR[91,3] = PR[90,3] + 24.578;
   1:L PR[91] R[100]mm/sec CNT100;
   1:  PR[91,1] = PR[90,1] + 1.116;
   1:  PR[91,2] = PR[90,2] + 12.598;
   1:  PR[91,3] = PR[90,3] + 24.590;
   1:L PR[91] R[100]mm/sec CNT100;
   1:  PR[91,1] = PR[90,1] + 0.646;
   1:  PR[91,2] = PR[90,2] + 12.420;
   1:  PR[91,3] = PR[90,3] + 24.594;
   1:L PR[91] R[100]mm/sec CNT100;
   1:  PR[91,1] = PR[90,1] + 0.152;
   1:  PR[91,2] = PR[90,2] + 12.326;
   1:  PR[91,3] = PR[90,3] + 24.597;
   1:L PR[91] R[100]mm/sec CNT100;
   1:  PR[91,1] = PR[90,1] + -0.345;
   1:  PR[91,2] = PR[90,2] + 12.324;
   1:  PR[91,3] = PR[90,3] + 24.601;
   1:L PR[91] R[100]mm/sec CNT100;
   1:  PR[91,1] = PR[90,1] + -0.829;
   1:  PR[91,2] = PR[90,2] + 12.403;
   1:  PR[91,3] = PR[90,3] + 24.605;
   1:L PR[91] R[100]mm/sec CNT100;
   1:  PR[91,1] = PR[90,1] + -1.149;
   1:  PR[91,2] = PR[90,2] + 12.512;
   1:  PR[91,3] = PR[90,3] + 24.608;
   1:L PR[91] R[100]mm/sec CNT100;
   1:  PR[91,1] = PR[90,1] + -1.308;
   1:  PR[91,2] = PR[90,2] + 12.573;
   1:  PR[91,3] = PR[90,3] + 24.611;
   1:L PR[91] R[100]mm/sec CNT100;
   1:  PR[91,1] = PR[90,1] + -1.734;
   1:  PR[91,2] = PR[90,2] + 12.808;
   1:  PR[91,3] = PR[90,3] + 24.612;
   1:L PR[91] R[100]mm/sec CNT100;
   1:  PR[91,1] = PR[90,1] + -2.098;
   1:  PR[91,2] = PR[90,2] + 13.097;
   1:  PR[91,3] = PR[90,3] + 24.616;
   1:L PR[91] R[100]mm/sec CNT100;
   1:  PR[91,1] = PR[90,1] + -3.024;
   1:  PR[91,2] = PR[90,2] + 13.899;
   1:  PR[91,3] = PR[90,3] + 24.619;
   1:L PR[91] R[100]mm/sec CNT100;
   1:  PR[91,1] = PR[90,1] + -3.799;
   1:  PR[91,2] = PR[90,2] + 14.492;
   1:  PR[91,3] = PR[90,3] + 24.628;
   1:L PR[91] R[100]mm/sec CNT100;
   1:  PR[91,1] = PR[90,1] + -4.609;
   1:  PR[91,2] = PR[90,2] + 15.046;
   1:  PR[91,3] = PR[90,3] + 24.635;
   1:L PR[91] R[100]mm/sec CNT100;
   1:  PR[91,1] = PR[90,1] + -5.449;
   1:  PR[91,2] = PR[90,2] + 15.558;
   1:  PR[91,3] = PR[90,3] + 24.642;
   1:L PR[91] R[100]mm/sec CNT100;
   1:  PR[91,1] = PR[90,1] + -6.316;
   1:  PR[91,2] = PR[90,2] + 16.028;
   1:  PR[91,3] = PR[90,3] + 24.649;
   1:L PR[91] R[100]mm/sec CNT100;
   1:  PR[91,1] = PR[90,1] + -7.209;
   1:  PR[91,2] = PR[90,2] + 16.454;
   1:  PR[91,3] = PR[90,3] + 24.657;
   1:L PR[91] R[100]mm/sec CNT100;
   1:  PR[91,1] = PR[90,1] + -8.123;
   1:  PR[91,2] = PR[90,2] + 16.835;
   1:  PR[91,3] = PR[90,3] + 24.664;
   1:L PR[91] R[100]mm/sec CNT100;
   1:  PR[91,1] = PR[90,1] + -9.057;
   1:  PR[91,2] = PR[90,2] + 17.169;
   1:  PR[91,3] = PR[90,3] + 24.671;
   1:L PR[91] R[100]mm/sec CNT100;
   1:  PR[91,1] = PR[90,1] + -10.007;
   1:  PR[91,2] = PR[90,2] + 17.456;
   1:  PR[91,3] = PR[90,3] + 24.678;
   1:L PR[91] R[100]mm/sec CNT100;
   1:  PR[91,1] = PR[90,1] + -10.972;
   1:  PR[91,2] = PR[90,2] + 17.693;
   1:  PR[91,3] = PR[90,3] + 24.686;
   1:L PR[91] R[100]mm/sec CNT100;
   1:  PR[91,1] = PR[90,1] + -11.948;
   1:  PR[91,2] = PR[90,2] + 17.883;
   1:  PR[91,3] = PR[90,3] + 24.693;
   1:L PR[91] R[100]mm/sec CNT100;
   1:  PR[91,1] = PR[90,1] + -12.933;
   1:  PR[91,2] = PR[90,2] + 18.023;
   1:  PR[91,3] = PR[90,3] + 24.700;
   1:L PR[91] R[100]mm/sec CNT100;
   1:  PR[91,1] = PR[90,1] + -13.924;
   1:  PR[91,2] = PR[90,2] + 18.116;
   1:  PR[91,3] = PR[90,3] + 24.707;
   1:L PR[91] R[100]mm/sec CNT100;
   1:  PR[91,1] = PR[90,1] + -14.874;
   1:  PR[91,2] = PR[90,2] + 18.160;
   1:  PR[91,3] = PR[90,3] + 24.715;
   1:L PR[91] R[100]mm/sec CNT100;
   1:  PR[91,1] = PR[90,1] + -15.912;
   1:  PR[91,2] = PR[90,2] + 18.156;
   1:  PR[91,3] = PR[90,3] + 24.722;
   1:L PR[91] R[100]mm/sec CNT100;
   1:  PR[91,1] = PR[90,1] + -16.802;
   1:  PR[91,2] = PR[90,2] + 18.110;
   1:  PR[91,3] = PR[90,3] + 24.729;
   1:L PR[91] R[100]mm/sec CNT100;
   1:  PR[91,1] = PR[90,1] + -17.888;
   1:  PR[91,2] = PR[90,2] + 18.001;
   1:  PR[91,3] = PR[90,3] + 24.736;
   1:L PR[91] R[100]mm/sec CNT100;
   1:  PR[91,1] = PR[90,1] + -18.708;
   1:  PR[91,2] = PR[90,2] + 17.879;
   1:  PR[91,3] = PR[90,3] + 24.744;
   1:L PR[91] R[100]mm/sec CNT100;
   1:  PR[91,1] = PR[90,1] + -19.829;
   1:  PR[91,2] = PR[90,2] + 17.656;
   1:  PR[91,3] = PR[90,3] + 24.750;
   1:L PR[91] R[100]mm/sec CNT100;
   1:  PR[91,1] = PR[90,1] + -20.572;
   1:  PR[91,2] = PR[90,2] + 17.470;
   1:  PR[91,3] = PR[90,3] + 24.758;
   1:L PR[91] R[100]mm/sec CNT100;
   1:  PR[91,1] = PR[90,1] + -21.714;
   1:  PR[91,2] = PR[90,2] + 17.125;
   1:  PR[91,3] = PR[90,3] + 24.764;
   1:L PR[91] R[100]mm/sec CNT100;
   1:  PR[91,1] = PR[90,1] + -22.378;
   1:  PR[91,2] = PR[90,2] + 16.889;
   1:  PR[91,3] = PR[90,3] + 24.772;
   1:L PR[91] R[100]mm/sec CNT100;
   1:  PR[91,1] = PR[90,1] + -23.529;
   1:  PR[91,2] = PR[90,2] + 16.415;
   1:  PR[91,3] = PR[90,3] + 24.778;
   1:L PR[91] R[100]mm/sec CNT100;
   1:  PR[91,1] = PR[90,1] + -24.117;
   1:  PR[91,2] = PR[90,2] + 16.139;
   1:  PR[91,3] = PR[90,3] + 24.787;
   1:L PR[91] R[100]mm/sec CNT100;
   1:  PR[91,1] = PR[90,1] + -24.683;
   1:  PR[91,2] = PR[90,2] + 15.851;
   1:  PR[91,3] = PR[90,3] + 24.791;
   1:L PR[91] R[100]mm/sec CNT100;
   1:  PR[91,1] = PR[90,1] + -25.285;
   1:  PR[91,2] = PR[90,2] + 15.519;
   1:  PR[91,3] = PR[90,3] + 24.796;
   1:L PR[91] R[100]mm/sec CNT100;
   1:  PR[91,1] = PR[90,1] + -25.928;
   1:  PR[91,2] = PR[90,2] + 15.131;
   1:  PR[91,3] = PR[90,3] + 24.801;
   1:L PR[91] R[100]mm/sec CNT100;
   1:  PR[91,1] = PR[90,1] + -26.904;
   1:  PR[91,2] = PR[90,2] + 14.477;
   1:  PR[91,3] = PR[90,3] + 24.806;
   1:L PR[91] R[100]mm/sec CNT100;
   1:  PR[91,1] = PR[90,1] + -27.548;
   1:  PR[91,2] = PR[90,2] + 13.993;
   1:  PR[91,3] = PR[90,3] + 24.815;
   1:L PR[91] R[100]mm/sec CNT100;
   1:  PR[91,1] = PR[90,1] + -28.335;
   1:  PR[91,2] = PR[90,2] + 13.342;
   1:  PR[91,3] = PR[90,3] + 24.821;
   1:L PR[91] R[100]mm/sec CNT100;
   1:  PR[91,1] = PR[90,1] + -28.966;
   1:  PR[91,2] = PR[90,2] + 12.761;
   1:  PR[91,3] = PR[90,3] + 24.828;
   1:L PR[91] R[100]mm/sec CNT100;
   1:  PR[91,1] = PR[90,1] + -29.601;
   1:  PR[91,2] = PR[90,2] + 12.117;
   1:  PR[91,3] = PR[90,3] + 24.835;
   1:L PR[91] R[100]mm/sec CNT100;
   1:  PR[91,1] = PR[90,1] + -30.187;
   1:  PR[91,2] = PR[90,2] + 11.456;
   1:  PR[91,3] = PR[90,3] + 24.841;
   1:L PR[91] R[100]mm/sec CNT100;
   1:  PR[91,1] = PR[90,1] + -30.737;
   1:  PR[91,2] = PR[90,2] + 10.769;
   1:  PR[91,3] = PR[90,3] + 24.848;
   1:L PR[91] R[100]mm/sec CNT100;
   1:  PR[91,1] = PR[90,1] + -31.250;
   1:  PR[91,2] = PR[90,2] + 10.056;
   1:  PR[91,3] = PR[90,3] + 24.854;
   1:L PR[91] R[100]mm/sec CNT100;
   1:  PR[91,1] = PR[90,1] + -31.726;
   1:  PR[91,2] = PR[90,2] + 9.321;
   1:  PR[91,3] = PR[90,3] + 24.861;
   1:L PR[91] R[100]mm/sec CNT100;
   1:  PR[91,1] = PR[90,1] + -32.163;
   1:  PR[91,2] = PR[90,2] + 8.566;
   1:  PR[91,3] = PR[90,3] + 24.867;
   1:L PR[91] R[100]mm/sec CNT100;
   1:  PR[91,1] = PR[90,1] + -32.562;
   1:  PR[91,2] = PR[90,2] + 7.796;
   1:  PR[91,3] = PR[90,3] + 24.873;
   1:L PR[91] R[100]mm/sec CNT100;
   1:  PR[91,1] = PR[90,1] + -32.920;
   1:  PR[91,2] = PR[90,2] + 7.016;
   1:  PR[91,3] = PR[90,3] + 24.880;
   1:L PR[91] R[100]mm/sec CNT100;
   1:  PR[91,1] = PR[90,1] + -33.238;
   1:  PR[91,2] = PR[90,2] + 6.231;
   1:  PR[91,3] = PR[90,3] + 24.886;
   1:L PR[91] R[100]mm/sec CNT100;
   1:  PR[91,1] = PR[90,1] + -33.513;
   1:  PR[91,2] = PR[90,2] + 5.442;
   1:  PR[91,3] = PR[90,3] + 24.892;
   1:L PR[91] R[100]mm/sec CNT100;
   1:  PR[91,1] = PR[90,1] + -33.747;
   1:  PR[91,2] = PR[90,2] + 4.648;
   1:  PR[91,3] = PR[90,3] + 24.898;
   1:L PR[91] R[100]mm/sec CNT100;
   1:  PR[91,1] = PR[90,1] + -33.938;
   1:  PR[91,2] = PR[90,2] + 3.847;
   1:  PR[91,3] = PR[90,3] + 24.904;
   1:L PR[91] R[100]mm/sec CNT100;
   1:  PR[91,1] = PR[90,1] + -34.088;
   1:  PR[91,2] = PR[90,2] + 3.032;
   1:  PR[91,3] = PR[90,3] + 24.910;
   1:L PR[91] R[100]mm/sec CNT100;
   1:  PR[91,1] = PR[90,1] + -34.195;
   1:  PR[91,2] = PR[90,2] + 2.194;
   1:  PR[91,3] = PR[90,3] + 24.916;
   1:L PR[91] R[100]mm/sec CNT100;
   1:  PR[91,1] = PR[90,1] + -34.259;
   1:  PR[91,2] = PR[90,2] + 1.328;
   1:  PR[91,3] = PR[90,3] + 24.923;
   1:L PR[91] R[100]mm/sec CNT100;
   1:  PR[91,1] = PR[90,1] + -34.282;
   1:  PR[91,2] = PR[90,2] + 0.428;
   1:  PR[91,3] = PR[90,3] + 24.929;
   1:L PR[91] R[100]mm/sec CNT100;
   1:  PR[91,1] = PR[90,1] + -34.259;
   1:  PR[91,2] = PR[90,2] + -0.473;
   1:  PR[91,3] = PR[90,3] + 24.936;
   1:L PR[91] R[100]mm/sec CNT100;
   1:  PR[91,1] = PR[90,1] + -34.195;
   1:  PR[91,2] = PR[90,2] + -1.339;
   1:  PR[91,3] = PR[90,3] + 24.942;
   1:L PR[91] R[100]mm/sec CNT100;
   1:  PR[91,1] = PR[90,1] + -34.088;
   1:  PR[91,2] = PR[90,2] + -2.176;
   1:  PR[91,3] = PR[90,3] + 24.948;
   1:L PR[91] R[100]mm/sec CNT100;
   1:  PR[91,1] = PR[90,1] + -33.938;
   1:  PR[91,2] = PR[90,2] + -2.992;
   1:  PR[91,3] = PR[90,3] + 24.955;
   1:L PR[91] R[100]mm/sec CNT100;
   1:  PR[91,1] = PR[90,1] + -33.747;
   1:  PR[91,2] = PR[90,2] + -3.793;
   1:  PR[91,3] = PR[90,3] + 24.961;
   1:L PR[91] R[100]mm/sec CNT100;
   1:  PR[91,1] = PR[90,1] + -33.513;
   1:  PR[91,2] = PR[90,2] + -4.587;
   1:  PR[91,3] = PR[90,3] + 24.967;
   1:L PR[91] R[100]mm/sec CNT100;
   1:  PR[91,1] = PR[90,1] + -33.238;
   1:  PR[91,2] = PR[90,2] + -5.376;
   1:  PR[91,3] = PR[90,3] + 24.973;
   1:L PR[91] R[100]mm/sec CNT100;
   1:  PR[91,1] = PR[90,1] + -32.920;
   1:  PR[91,2] = PR[90,2] + -6.161;
   1:  PR[91,3] = PR[90,3] + 24.979;
   1:L PR[91] R[100]mm/sec CNT100;
   1:  PR[91,1] = PR[90,1] + -32.562;
   1:  PR[91,2] = PR[90,2] + -6.941;
   1:  PR[91,3] = PR[90,3] + 24.985;
   1:L PR[91] R[100]mm/sec CNT100;
   1:  PR[91,1] = PR[90,1] + -32.163;
   1:  PR[91,2] = PR[90,2] + -7.711;
   1:  PR[91,3] = PR[90,3] + 24.991;
   1:L PR[91] R[100]mm/sec CNT100;
   1:  PR[91,1] = PR[90,1] + -31.726;
   1:  PR[91,2] = PR[90,2] + -8.466;
   1:  PR[91,3] = PR[90,3] + 24.998;
   1:L PR[91] R[100]mm/sec CNT100;
   1:  PR[91,1] = PR[90,1] + -31.250;
   1:  PR[91,2] = PR[90,2] + -9.201;
   1:  PR[91,3] = PR[90,3] + 25.004;
